LIN {X 0,Y 264.85,Z 561.545,A -85,B 0,C 180,E1 -18192.841,E2 -18192.841} C_VEL
LIN {X 0,Y 265.492,Z 550.133,A -85,B 0,C 180,E1 -18194.761,E2 -18194.761} C_VEL
LIN {X 0,Y 266.161,Z 538.928,A -85,B 0,C 180,E1 -18196.293,E2 -18196.293} C_VEL
LIN {X 0,Y 267.031,Z 524.888,A -85,B 0,C 180,E1 -18197.816,E2 -18197.816} C_VEL
LIN {X 0,Y 267.504,Z 510.963,A -85,B 0,C 180,E1 -18198.948,E2 -18198.948} C_VEL
LIN {X 0,Y 267.86,Z 496.922,A -85,B 0,C 180,E1 -18199.767,E2 -18199.767} C_VEL
LIN {X 0,Y 269.082,Z 449.76,A -85,B 0,C 180,E1 -18201.707,E2 -18201.707} C_VEL
LIN {X 0,Y 269.543,Z 437.735,A -85,B 0,C 180,E1 -18202.197,E2 -18202.197} C_VEL
LIN {X 0,Y 263.446,Z 416.884,A -85,B 0,C 180,E1 -18203.35,E2 -18203.35} C_VEL
LIN {X 0,Y 263.229,Z 415.845,A -85,B 0,C 180,E1 -18203.609,E2 -18203.609} C_VEL
LIN {X 0,Y 263.152,Z 415.684,A -85,B 0,C 180,E1 -18208.197,E2 -18208.197} C_VEL
LIN {X 0,Y 263.129,Z 415.701,A -85,B 0,C 180,E1 -18212.289,E2 -18212.289} C_VEL
LIN {X 0,Y 263.183,Z 415.698,A -85,B 0,C 180,E1 -18216.763,E2 -18216.763} C_VEL
LIN {X 0,Y 263.126,Z 415.699,A -85,B 0,C 180,E1 -18221.594,E2 -18221.594} C_VEL
LIN {X 0,Y 263.161,Z 415.973,A -85,B 0,C 180,E1 -18223.119,E2 -18223.119} C_VEL
LIN {X 0,Y 267.955,Z 428.767,A -85,B 0,C 180,E1 -18227.005,E2 -18227.005} C_VEL
LIN {X 0,Y 272.039,Z 441.377,A -85,B 0,C 180,E1 -18230.442,E2 -18230.442} C_VEL
LIN {X 0,Y 275.291,Z 453.83,A -85,B 0,C 180,E1 -18233.539,E2 -18233.539} C_VEL
LIN {X 0,Y 277.381,Z 463.477,A -85,B 0,C 180,E1 -18235.787,E2 -18235.787} C_VEL
LIN {X 0,Y 277.002,Z 468.199,A -85,B 0,C 180,E1 -18236.672,E2 -18236.672} C_VEL
LIN {X 0,Y 274.845,Z 486.292,A -85,B 0,C 180,E1 -18239.872,E2 -18239.872} C_VEL
LIN {X 0,Y 274.77,Z 488.523,A -85,B 0,C 180,E1 -18240.174,E2 -18240.174} C_VEL
LIN {X 0,Y 279.262,Z 521.145,A -85,B 0,C 180,E1 -18241.646,E2 -18241.646} C_VEL
LIN {X 0,Y 279.718,Z 525.519,A -85,B 0,C 180,E1 -18241.821,E2 -18241.821} C_VEL
LIN {X 0,Y 277.38,Z 599.883,A -85,B 0,C 180,E1 -18243.73,E2 -18243.73} C_VEL
LIN {X 0,Y 276.41,Z 612.805,A -85,B 0,C 180,E1 -18244.289,E2 -18244.289} C_VEL
LIN {X 0,Y 275.09,Z 625.722,A -85,B 0,C 180,E1 -18245.169,E2 -18245.169} C_VEL
LIN {X 0,Y 273.45,Z 638.017,A -85,B 0,C 180,E1 -18246.323,E2 -18246.323} C_VEL
LIN {X 0,Y 271.782,Z 648.339,A -85,B 0,C 180,E1 -18247.578,E2 -18247.578} C_VEL
LIN {X 0,Y 269.838,Z 658.927,A -85,B 0,C 180,E1 -18249.215,E2 -18249.215} C_VEL
LIN {X 0,Y 267.978,Z 668.621,A -85,B 0,C 180,E1 -18251.099,E2 -18251.099} C_VEL
LIN {X 0,Y 266.264,Z 677.005,A -85,B 0,C 180,E1 -18253.122,E2 -18253.122} C_VEL
LIN {X 0,Y 264.551,Z 684.486,A -85,B 0,C 180,E1 -18255.382,E2 -18255.382} C_VEL
LIN {X 0,Y 263.269,Z 690.488,A -85,B 0,C 180,E1 -18257.669,E2 -18257.669} C_VEL
LIN {X 0,Y 262.296,Z 695.236,A -85,B 0,C 180,E1 -18259.97,E2 -18259.97} C_VEL
LIN {X 0,Y 261.682,Z 698.867,A -85,B 0,C 180,E1 -18262.283,E2 -18262.283} C_VEL
LIN {X 0,Y 261.26,Z 701.355,A -85,B 0,C 180,E1 -18264.454,E2 -18264.454} C_VEL
LIN {X 0,Y 261.111,Z 703.163,A -85,B 0,C 180,E1 -18266.914,E2 -18266.914} C_VEL
LIN {X 0,Y 261.076,Z 704.013,A -85,B 0,C 180,E1 -18270,E2 -18270} C_VEL
LIN {X 0,Y 261.054,Z 703.816,A -85,B 0,C 180,E1 -18271.543,E2 -18271.543} C_VEL
LIN {X 0,Y 261.109,Z 703.224,A -85,B 0,C 180,E1 -18273.086,E2 -18273.086} C_VEL
LIN {X 0,Y 261.244,Z 701.499,A -85,B 0,C 180,E1 -18275.509,E2 -18275.509} C_VEL
LIN {X 0,Y 261.808,Z 697.975,A -85,B 0,C 180,E1 -18278.491,E2 -18278.491} C_VEL
LIN {X 0,Y 262.551,Z 694.043,A -85,B 0,C 180,E1 -18280.8,E2 -18280.8} C_VEL
LIN {X 0,Y 263.619,Z 688.947,A -85,B 0,C 180,E1 -18283.098,E2 -18283.098} C_VEL
LIN {X 0,Y 265.02,Z 682.524,A -85,B 0,C 180,E1 -18285.378,E2 -18285.378} C_VEL
LIN {X 0,Y 266.866,Z 674.544,A -85,B 0,C 180,E1 -18287.63,E2 -18287.63} C_VEL
LIN {X 0,Y 268.529,Z 666.026,A -85,B 0,C 180,E1 -18289.575,E2 -18289.575} C_VEL
LIN {X 0,Y 270.323,Z 656.341,A -85,B 0,C 180,E1 -18291.345,E2 -18291.345} C_VEL
LIN {X 0,Y 272.405,Z 645.045,A -85,B 0,C 180,E1 -18292.969,E2 -18292.969} C_VEL
LIN {X 0,Y 274.123,Z 633.931,A -85,B 0,C 180,E1 -18294.218,E2 -18294.218} C_VEL
LIN {X 0,Y 275.628,Z 621.337,A -85,B 0,C 180,E1 -18295.284,E2 -18295.284} C_VEL
LIN {X 0,Y 276.909,Z 608.091,A -85,B 0,C 180,E1 -18296.066,E2 -18296.066} C_VEL
LIN {X 0,Y 277.692,Z 594.677,A -85,B 0,C 180,E1 -18296.542,E2 -18296.542} C_VEL
LIN {X 0,Y 279.693,Z 524.43,A -85,B 0,C 180,E1 -18298.337,E2 -18298.337} C_VEL
LIN {X 0,Y 275.48,Z 492.805,A -85,B 0,C 180,E1 -18299.737,E2 -18299.737} C_VEL
LIN {X 0,Y 274.779,Z 487.724,A -85,B 0,C 180,E1 -18300.016,E2 -18300.016} C_VEL
LIN {X 0,Y 277.378,Z 465.897,A -85,B 0,C 180,E1 -18303.878,E2 -18303.878} C_VEL
LIN {X 0,Y 277.535,Z 464.171,A -85,B 0,C 180,E1 -18304.208,E2 -18304.208} C_VEL
LIN {X 0,Y 275.261,Z 453.468,A -85,B 0,C 180,E1 -18306.688,E2 -18306.688} C_VEL
LIN {X 0,Y 272.521,Z 442.891,A -85,B 0,C 180,E1 -18309.315,E2 -18309.315} C_VEL
LIN {X 0,Y 268.936,Z 431.503,A -85,B 0,C 180,E1 -18312.417,E2 -18312.417} C_VEL
LIN {X 0,Y 265.144,Z 421.282,A -85,B 0,C 180,E1 -18315.379,E2 -18315.379} C_VEL
LIN {X 0,Y 263.143,Z 415.913,A -85,B 0,C 180,E1 -18317.074,E2 -18317.074} C_VEL
LIN {X 0,Y 263.115,Z 415.714,A -85,B 0,C 180,E1 -18320.771,E2 -18320.771} C_VEL
LIN {X 0,Y 263.16,Z 415.701,A -85,B 0,C 180,E1 -18324.017,E2 -18324.017} C_VEL
LIN {X 0,Y 263.111,Z 415.698,A -85,B 0,C 180,E1 -18327.315,E2 -18327.315} C_VEL
LIN {X 0,Y 262.472,Z 415.792,A -85,B 0,C 180,E1 -18328.594,E2 -18328.594} C_VEL
LIN {X 0,Y 259.622,Z 416.159,A -85,B 0,C 180,E1 -18330.677,E2 -18330.677} C_VEL
LIN {X 0,Y 257.197,Z 416.463,A -85,B 0,C 180,E1 -18332.372,E2 -18332.372} C_VEL
LIN {X 0,Y 256.172,Z 416.58,A -85,B 0,C 180,E1 -18333.686,E2 -18333.686} C_VEL
LIN {X 0,Y 256.098,Z 416.584,A -85,B 0,C 180,E1 -18334.132,E2 -18334.132} C_VEL
LIN {X 0,Y 256.074,Z 416.57,A -85,B 0,C 180,E1 -18337.404,E2 -18337.404} C_VEL
LIN {X 0,Y 256.111,Z 416.568,A -85,B 0,C 180,E1 -18340.774,E2 -18340.774} C_VEL
LIN {X 0,Y 256.216,Z 416.56,A -85,B 0,C 180,E1 -18344.08,E2 -18344.08} C_VEL
LIN {X 0,Y 256.277,Z 416.532,A -85,B 0,C 180,E1 -18348.932,E2 -18348.932} C_VEL
LIN {X 0,Y 256.493,Z 416.535,A -85,B 0,C 180,E1 -18352.125,E2 -18352.125} C_VEL
LIN {X 0,Y 256.451,Z 416.518,A -85,B 0,C 180,E1 -18356.858,E2 -18356.858} C_VEL
LIN {X 0,Y 256.699,Z 416.509,A -85,B 0,C 180,E1 -18358.431,E2 -18358.431} C_VEL
LIN {X 0,Y 256.697,Z 416.481,A -85,B 0,C 180,E1 -18361.569,E2 -18361.569} C_VEL
LIN {X 0,Y 256.458,Z 416.539,A -85,B 0,C 180,E1 -18366.293,E2 -18366.293} C_VEL
LIN {X 0,Y 256.405,Z 416.515,A -85,B 0,C 180,E1 -18369.466,E2 -18369.466} C_VEL
LIN {X 0,Y 256.207,Z 416.564,A -85,B 0,C 180,E1 -18374.293,E2 -18374.293} C_VEL
LIN {X 0,Y 256.142,Z 416.553,A -85,B 0,C 180,E1 -18377.567,E2 -18377.567} C_VEL
LIN {X 0,Y 256.121,Z 416.572,A -85,B 0,C 180,E1 -18381.097,E2 -18381.097} C_VEL
LIN {X 0,Y 256.084,Z 416.578,A -85,B 0,C 180,E1 -18385.087,E2 -18385.087} C_VEL
LIN {X 0,Y 256.078,Z 416.564,A -85,B 0,C 180,E1 -18388.569,E2 -18388.569} C_VEL
LIN {X 0,Y 256.072,Z 416.588,A -85,B 0,C 180,E1 -18391.699,E2 -18391.699} C_VEL
LIN {X 0,Y 256.081,Z 416.57,A -85,B 0,C 180,E1 -18395.193,E2 -18395.193} C_VEL
LIN {X 0,Y 256.107,Z 416.584,A -85,B 0,C 180,E1 -18397.268,E2 -18397.268} C_VEL
LIN {X 0,Y 256.018,Z 416.527,A -85,B 0,C 180,E1 -18401.211,E2 -18401.211} C_VEL
LIN {X 0,Y 256.034,Z 416.594,A -85,B 0,C 180,E1 -18405.536,E2 -18405.536} C_VEL
LIN {X 0,Y 256.023,Z 416.717,A -85,B 0,C 180,E1 -18409.354,E2 -18409.354} C_VEL
LIN {X 0,Y 256.297,Z 417.843,A -85,B 0,C 180,E1 -18409.759,E2 -18409.759} C_VEL
LIN {X 0,Y 259.881,Z 424.387,A -85,B 0,C 180,E1 -18411.31,E2 -18411.31} C_VEL
LIN {X 0,Y 263.321,Z 435.836,A -85,B 0,C 180,E1 -18413.197,E2 -18413.197} C_VEL
LIN {X 0,Y 267.896,Z 451.956,A -85,B 0,C 180,E1 -18415.612,E2 -18415.612} C_VEL
LIN {X 0,Y 268.711,Z 455.376,A -85,B 0,C 180,E1 -18416.083,E2 -18416.083} C_VEL
LIN {X 0,Y 268.725,Z 480.622,A -85,B 0,C 180,E1 -18418.681,E2 -18418.681} C_VEL
LIN {X 0,Y 268.671,Z 489.032,A -85,B 0,C 180,E1 -18419.496,E2 -18419.496} C_VEL
LIN {X 0,Y 271.982,Z 520.346,A -85,B 0,C 180,E1 -18420.837,E2 -18420.837} C_VEL
LIN {X 0,Y 272.827,Z 533.578,A -85,B 0,C 180,E1 -18421.325,E2 -18421.325} C_VEL
LIN {X 0,Y 270.595,Z 602.971,A -85,B 0,C 180,E1 -18423.122,E2 -18423.122} C_VEL
LIN {X 0,Y 269.625,Z 616.536,A -85,B 0,C 180,E1 -18423.697,E2 -18423.697} C_VEL
LIN {X 0,Y 268.323,Z 628.565,A -85,B 0,C 180,E1 -18424.498,E2 -18424.498} C_VEL
LIN {X 0,Y 266.64,Z 641.245,A -85,B 0,C 180,E1 -18425.679,E2 -18425.679} C_VEL
LIN {X 0,Y 264.897,Z 651.794,A -85,B 0,C 180,E1 -18426.962,E2 -18426.962} C_VEL
LIN {X 0,Y 262.808,Z 662.552,A -85,B 0,C 180,E1 -18428.631,E2 -18428.631} C_VEL
LIN {X 0,Y 260.829,Z 672.425,A -85,B 0,C 180,E1 -18430.574,E2 -18430.574} C_VEL
LIN {X 0,Y 259.036,Z 680.818,A -85,B 0,C 180,E1 -18432.635,E2 -18432.635} C_VEL
LIN {X 0,Y 257.333,Z 688.353,A -85,B 0,C 180,E1 -18434.962,E2 -18434.962} C_VEL
LIN {X 0,Y 256.017,Z 694.402,A -85,B 0,C 180,E1 -18437.314,E2 -18437.314} C_VEL
LIN {X 0,Y 255.09,Z 699.178,A -85,B 0,C 180,E1 -18439.683,E2 -18439.683} C_VEL
LIN {X 0,Y 254.443,Z 702.823,A -85,B 0,C 180,E1 -18442.061,E2 -18442.061} C_VEL
LIN {X 0,Y 254.126,Z 705.608,A -85,B 0,C 180,E1 -18444.625,E2 -18444.625} C_VEL
LIN {X 0,Y 254.03,Z 707.114,A -85,B 0,C 180,E1 -18446.828,E2 -18446.828} C_VEL
LIN {X 0,Y 254.025,Z 707.724,A -85,B 0,C 180,E1 -18448.414,E2 -18448.414} C_VEL
LIN {X 0,Y 254.065,Z 707.939,A -85,B 0,C 180,E1 -18450,E2 -18450} C_VEL
LIN {X 0,Y 254.067,Z 707.715,A -85,B 0,C 180,E1 -18451.585,E2 -18451.585} C_VEL
LIN {X 0,Y 254.054,Z 707.099,A -85,B 0,C 180,E1 -18453.171,E2 -18453.171} C_VEL
LIN {X 0,Y 254.134,Z 705.563,A -85,B 0,C 180,E1 -18455.394,E2 -18455.394} C_VEL
LIN {X 0,Y 254.451,Z 702.782,A -85,B 0,C 180,E1 -18457.938,E2 -18457.938} C_VEL
LIN {X 0,Y 255.092,Z 699.121,A -85,B 0,C 180,E1 -18460.316,E2 -18460.316} C_VEL
LIN {X 0,Y 256.021,Z 694.331,A -85,B 0,C 180,E1 -18462.686,E2 -18462.686} C_VEL
LIN {X 0,Y 257.345,Z 688.269,A -85,B 0,C 180,E1 -18465.037,E2 -18465.037} C_VEL
LIN {X 0,Y 259.024,Z 680.707,A -85,B 0,C 180,E1 -18467.365,E2 -18467.365} C_VEL
LIN {X 0,Y 260.837,Z 672.247,A -85,B 0,C 180,E1 -18469.431,E2 -18469.431} C_VEL
LIN {X 0,Y 262.817,Z 662.368,A -85,B 0,C 180,E1 -18471.367,E2 -18471.367} C_VEL
LIN {X 0,Y 264.865,Z 651.56,A -85,B 0,C 180,E1 -18473.04,E2 -18473.04} C_VEL
LIN {X 0,Y 266.889,Z 639.21,A -85,B 0,C 180,E1 -18474.503,E2 -18474.503} C_VEL
LIN {X 0,Y 267.731,Z 633.457,A -85,B 0,C 180,E1 -18475.094,E2 -18475.094} C_VEL
LIN {X 0,Y 272.517,Z 622.346,A -85,B 0,C 180,E1 -18477.243,E2 -18477.243} C_VEL
LIN {X 0,Y 277.231,Z 610.736,A -85,B 0,C 180,E1 -18479.001,E2 -18479.001} C_VEL
LIN {X 0,Y 281.94,Z 597.942,A -85,B 0,C 180,E1 -18480.524,E2 -18480.524} C_VEL
LIN {X 0,Y 285.924,Z 585.491,A -85,B 0,C 180,E1 -18481.695,E2 -18481.695} C_VEL
LIN {X 0,Y 289.914,Z 571.079,A -85,B 0,C 180,E1 -18482.744,E2 -18482.744} C_VEL
LIN {X 0,Y 293.532,Z 553.924,A -85,B 0,C 180,E1 -18483.688,E2 -18483.688} C_VEL
LIN {X 0,Y 296.227,Z 535.792,A -85,B 0,C 180,E1 -18484.52,E2 -18484.52} C_VEL
LIN {X 0,Y 297.419,Z 522.403,A -85,B 0,C 180,E1 -18485.437,E2 -18485.437} C_VEL
LIN {X 0,Y 298.17,Z 508.364,A -85,B 0,C 180,E1 -18486.705,E2 -18486.705} C_VEL
LIN {X 0,Y 298.597,Z 495.67,A -85,B 0,C 180,E1 -18488.12,E2 -18488.12} C_VEL
LIN {X 0,Y 298.719,Z 489.21,A -85,B 0,C 180,E1 -18488.995,E2 -18488.995} C_VEL
LIN {X 0,Y 297.581,Z 483.469,A -85,B 0,C 180,E1 -18490.746,E2 -18490.746} C_VEL
LIN {X 0,Y 296.387,Z 477.666,A -85,B 0,C 180,E1 -18493.445,E2 -18493.445} C_VEL
LIN {X 0,Y 296.175,Z 474.72,A -85,B 0,C 180,E1 -18495.573,E2 -18495.573} C_VEL
LIN {X 0,Y 296.767,Z 472.828,A -85,B 0,C 180,E1 -18498.053,E2 -18498.053} C_VEL
LIN {X 0,Y 298.296,Z 472.538,A -85,B 0,C 180,E1 -18500.496,E2 -18500.496} C_VEL
LIN {X 0,Y 300.271,Z 473.517,A -85,B 0,C 180,E1 -18502.516,E2 -18502.516} C_VEL
LIN {X 0,Y 302.602,Z 475.847,A -85,B 0,C 180,E1 -18504.379,E2 -18504.379} C_VEL
LIN {X 0,Y 304.246,Z 477.887,A -85,B 0,C 180,E1 -18505.466,E2 -18505.466} C_VEL
LIN {X 0,Y 299.441,Z 507.153,A -85,B 0,C 180,E1 -18506.881,E2 -18506.881} C_VEL
LIN {X 0,Y 297.506,Z 521.717,A -85,B 0,C 180,E1 -18507.742,E2 -18507.742} C_VEL
LIN {X 0,Y 295.036,Z 535.372,A -85,B 0,C 180,E1 -18508.795,E2 -18508.795} C_VEL
LIN {X 0,Y 292.316,Z 546.909,A -85,B 0,C 180,E1 -18509.944,E2 -18509.944} C_VEL
LIN {X 0,Y 289.223,Z 557.964,A -85,B 0,C 180,E1 -18511.32,E2 -18511.32} C_VEL
LIN {X 0,Y 285.591,Z 568.323,A -85,B 0,C 180,E1 -18512.918,E2 -18512.918} C_VEL
LIN {X 0,Y 282.305,Z 576.824,A -85,B 0,C 180,E1 -18514.535,E2 -18514.535} C_VEL
LIN {X 0,Y 278.49,Z 585.306,A -85,B 0,C 180,E1 -18516.58,E2 -18516.58} C_VEL
LIN {X 0,Y 274.934,Z 592.143,A -85,B 0,C 180,E1 -18518.638,E2 -18518.638} C_VEL
LIN {X 0,Y 271.125,Z 598.395,A -85,B 0,C 180,E1 -18521.094,E2 -18521.094} C_VEL
LIN {X 0,Y 267.32,Z 603.574,A -85,B 0,C 180,E1 -18523.975,E2 -18523.975} C_VEL
LIN {X 0,Y 264.813,Z 606.237,A -85,B 0,C 180,E1 -18526.181,E2 -18526.181} C_VEL
LIN {X 0,Y 263.333,Z 607.422,A -85,B 0,C 180,E1 -18527.672,E2 -18527.672} C_VEL
LIN {X 0,Y 260.7,Z 608.594,A -85,B 0,C 180,E1 -18530.692,E2 -18530.692} C_VEL
LIN {X 0,Y 259.67,Z 608.534,A -85,B 0,C 180,E1 -18532.223,E2 -18532.223} C_VEL
LIN {X 0,Y 258.912,Z 608.014,A -85,B 0,C 180,E1 -18533.767,E2 -18533.767} C_VEL
LIN {X 0,Y 258.281,Z 607.095,A -85,B 0,C 180,E1 -18535.318,E2 -18535.318} C_VEL
LIN {X 0,Y 257.555,Z 605.796,A -85,B 0,C 180,E1 -18536.872,E2 -18536.872} C_VEL
LIN {X 0,Y 256.743,Z 602.999,A -85,B 0,C 180,E1 -18539.216,E2 -18539.216} C_VEL
LIN {X 0,Y 256.327,Z 599.154,A -85,B 0,C 180,E1 -18541.571,E2 -18541.571} C_VEL
LIN {X 0,Y 256.161,Z 594.186,A -85,B 0,C 180,E1 -18543.933,E2 -18543.933} C_VEL
LIN {X 0,Y 256.322,Z 586.806,A -85,B 0,C 180,E1 -18546.692,E2 -18546.692} C_VEL
LIN {X 0,Y 256.735,Z 578.927,A -85,B 0,C 180,E1 -18549.056,E2 -18549.056} C_VEL
LIN {X 0,Y 257.298,Z 569.105,A -85,B 0,C 180,E1 -18551.422,E2 -18551.422} C_VEL
LIN {X 0,Y 257.907,Z 559.145,A -85,B 0,C 180,E1 -18553.393,E2 -18553.393} C_VEL
LIN {X 0,Y 258.623,Z 546.833,A -85,B 0,C 180,E1 -18555.364,E2 -18555.364} C_VEL
LIN {X 0,Y 259.376,Z 534.597,A -85,B 0,C 180,E1 -18556.935,E2 -18556.935} C_VEL
LIN {X 0,Y 260.126,Z 521.014,A -85,B 0,C 180,E1 -18558.305,E2 -18558.305} C_VEL
LIN {X 0,Y 260.522,Z 507.02,A -85,B 0,C 180,E1 -18559.361,E2 -18559.361} C_VEL
LIN {X 0,Y 260.898,Z 492.906,A -85,B 0,C 180,E1 -18560.109,E2 -18560.109} C_VEL
LIN {X 0,Y 262.036,Z 451.118,A -85,B 0,C 180,E1 -18561.899,E2 -18561.899} C_VEL
LIN {X 0,Y 262.46,Z 438.689,A -85,B 0,C 180,E1 -18562.423,E2 -18562.423} C_VEL
LIN {X 0,Y 256.376,Z 417.606,A -85,B 0,C 180,E1 -18563.616,E2 -18563.616} C_VEL
LIN {X 0,Y 256.189,Z 416.651,A -85,B 0,C 180,E1 -18563.928,E2 -18563.928} C_VEL
LIN {X 0,Y 256.094,Z 416.561,A -85,B 0,C 180,E1 -18568.577,E2 -18568.577} C_VEL
LIN {X 0,Y 256.076,Z 416.588,A -85,B 0,C 180,E1 -18571.702,E2 -18571.702} C_VEL
LIN {X 0,Y 256.083,Z 416.575,A -85,B 0,C 180,E1 -18575.193,E2 -18575.193} C_VEL
LIN {X 0,Y 256.115,Z 416.572,A -85,B 0,C 180,E1 -18577.271,E2 -18577.271} C_VEL
LIN {X 0,Y 256.129,Z 416.804,A -85,B 0,C 180,E1 -18581.83,E2 -18581.83} C_VEL
LIN {X 0,Y 260.412,Z 428.088,A -85,B 0,C 180,E1 -18585.437,E2 -18585.437} C_VEL
LIN {X 0,Y 263.748,Z 437.752,A -85,B 0,C 180,E1 -18588.255,E2 -18588.255} C_VEL
LIN {X 0,Y 266.799,Z 447.885,A -85,B 0,C 180,E1 -18590.994,E2 -18590.994} C_VEL
LIN {X 0,Y 269.972,Z 460.995,A -85,B 0,C 180,E1 -18594.251,E2 -18594.251} C_VEL
LIN {X 0,Y 270.983,Z 466.791,A -85,B 0,C 180,E1 -18595.577,E2 -18595.577} C_VEL
LIN {X 0,Y 268.545,Z 486.331,A -85,B 0,C 180,E1 -18599.096,E2 -18599.096} C_VEL
LIN {X 0,Y 268.429,Z 488.341,A -85,B 0,C 180,E1 -18599.388,E2 -18599.388} C_VEL
LIN {X 0,Y 273.023,Z 521.924,A -85,B 0,C 180,E1 -18600.961,E2 -18600.961} C_VEL
LIN {X 0,Y 273.425,Z 527.263,A -85,B 0,C 180,E1 -18601.165,E2 -18601.165} C_VEL
LIN {X 0,Y 270.974,Z 601.199,A -85,B 0,C 180,E1 -18603.111,E2 -18603.111} C_VEL
LIN {X 0,Y 269.893,Z 614.342,A -85,B 0,C 180,E1 -18603.725,E2 -18603.725} C_VEL
LIN {X 0,Y 268.431,Z 627.911,A -85,B 0,C 180,E1 -18604.717,E2 -18604.717} C_VEL
LIN {X 0,Y 266.728,Z 639.694,A -85,B 0,C 180,E1 -18605.895,E2 -18605.895} C_VEL
LIN {X 0,Y 264.759,Z 650.917,A -85,B 0,C 180,E1 -18607.362,E2 -18607.362} C_VEL
LIN {X 0,Y 262.814,Z 661.059,A -85,B 0,C 180,E1 -18609.043,E2 -18609.043} C_VEL
LIN {X 0,Y 260.802,Z 671.014,A -85,B 0,C 180,E1 -18611.133,E2 -18611.133} C_VEL
LIN {X 0,Y 258.816,Z 679.726,A -85,B 0,C 180,E1 -18613.434,E2 -18613.434} C_VEL
LIN {X 0,Y 257.152,Z 686.717,A -85,B 0,C 180,E1 -18615.761,E2 -18615.761} C_VEL
LIN {X 0,Y 255.936,Z 692.271,A -85,B 0,C 180,E1 -18618.115,E2 -18618.115} C_VEL
LIN {X 0,Y 255.028,Z 696.629,A -85,B 0,C 180,E1 -18620.483,E2 -18620.483} C_VEL
LIN {X 0,Y 254.627,Z 698.922,A -85,B 0,C 180,E1 -18622.068,E2 -18622.068} C_VEL
LIN {X 0,Y 254.168,Z 701.613,A -85,B 0,C 180,E1 -18624.526,E2 -18624.526} C_VEL
LIN {X 0,Y 254.012,Z 703.218,A -85,B 0,C 180,E1 -18626.828,E2 -18626.828} C_VEL
LIN {X 0,Y 253.967,Z 703.833,A -85,B 0,C 180,E1 -18628.414,E2 -18628.414} C_VEL
LIN {X 0,Y 253.984,Z 704.067,A -85,B 0,C 180,E1 -18630,E2 -18630} C_VEL
LIN {X 0,Y 253.966,Z 703.87,A -85,B 0,C 180,E1 -18631.586,E2 -18631.586} C_VEL
LIN {X 0,Y 254.01,Z 703.278,A -85,B 0,C 180,E1 -18633.172,E2 -18633.172} C_VEL
LIN {X 0,Y 254.135,Z 701.794,A -85,B 0,C 180,E1 -18635.394,E2 -18635.394} C_VEL
LIN {X 0,Y 254.564,Z 699.081,A -85,B 0,C 180,E1 -18637.935,E2 -18637.935} C_VEL
LIN {X 0,Y 255.267,Z 695.504,A -85,B 0,C 180,E1 -18640.309,E2 -18640.309} C_VEL
LIN {X 0,Y 256.273,Z 690.812,A -85,B 0,C 180,E1 -18642.674,E2 -18642.674} C_VEL
LIN {X 0,Y 257.587,Z 684.867,A -85,B 0,C 180,E1 -18645.023,E2 -18645.023} C_VEL
LIN {X 0,Y 259.401,Z 677.47,A -85,B 0,C 180,E1 -18647.339,E2 -18647.339} C_VEL
LIN {X 0,Y 261.344,Z 668.537,A -85,B 0,C 180,E1 -18649.557,E2 -18649.557} C_VEL
LIN {X 0,Y 263.281,Z 658.574,A -85,B 0,C 180,E1 -18651.534,E2 -18651.534} C_VEL
LIN {X 0,Y 265.401,Z 647.843,A -85,B 0,C 180,E1 -18653.198,E2 -18653.198} C_VEL
LIN {X 0,Y 267.435,Z 635.686,A -85,B 0,C 180,E1 -18654.657,E2 -18654.657} C_VEL
LIN {X 0,Y 268.983,Z 623.804,A -85,B 0,C 180,E1 -18655.746,E2 -18655.746} C_VEL
LIN {X 0,Y 270.248,Z 611.484,A -85,B 0,C 180,E1 -18656.55,E2 -18656.55} C_VEL
LIN {X 0,Y 271.224,Z 597.771,A -85,B 0,C 180,E1 -18657.123,E2 -18657.123} C_VEL
LIN {X 0,Y 273.395,Z 524.791,A -85,B 0,C 180,E1 -18659.038,E2 -18659.038} C_VEL
LIN {X 0,Y 269.172,Z 492.941,A -85,B 0,C 180,E1 -18660.5,E2 -18660.5} C_VEL
LIN {X 0,Y 268.473,Z 487.826,A -85,B 0,C 180,E1 -18660.779,E2 -18660.779} C_VEL
LIN {X 0,Y 270.976,Z 467.525,A -85,B 0,C 180,E1 -18664.418,E2 -18664.418} C_VEL
LIN {X 0,Y 270.801,Z 464.663,A -85,B 0,C 180,E1 -18665.044,E2 -18665.044} C_VEL
LIN {X 0,Y 267.934,Z 452.006,A -85,B 0,C 180,E1 -18668.102,E2 -18668.102} C_VEL
LIN {X 0,Y 265.472,Z 443.079,A -85,B 0,C 180,E1 -18670.437,E2 -18670.437} C_VEL
LIN {X 0,Y 261.856,Z 431.948,A -85,B 0,C 180,E1 -18673.559,E2 -18673.559} C_VEL
LIN {X 0,Y 257.599,Z 420.812,A -85,B 0,C 180,E1 -18676.994,E2 -18676.994} C_VEL
LIN {X 0,Y 256.112,Z 416.811,A -85,B 0,C 180,E1 -18678.33,E2 -18678.33} C_VEL
LIN {X 0,Y 256.068,Z 416.592,A -85,B 0,C 180,E1 -18680.857,E2 -18680.857} C_VEL
LIN {X 0,Y 256.082,Z 416.587,A -85,B 0,C 180,E1 -18684.807,E2 -18684.807} C_VEL
LIN {X 0,Y 256.08,Z 416.589,A -85,B 0,C 180,E1 -18688.57,E2 -18688.57} C_VEL
LIN {X 0,Y 256.088,Z 416.573,A -85,B 0,C 180,E1 -18692.19,E2 -18692.19} C_VEL
LIN {X 0,Y 256.098,Z 416.584,A -85,B 0,C 180,E1 -18694.132,E2 -18694.132} C_VEL
LIN {X 0,Y 255.446,Z 416.652,A -85,B 0,C 180,E1 -18695.445,E2 -18695.445} C_VEL
LIN {X 0,Y 252.574,Z 417.011,A -85,B 0,C 180,E1 -18697.585,E2 -18697.585} C_VEL
LIN {X 0,Y 250.136,Z 417.329,A -85,B 0,C 180,E1 -18699.328,E2 -18699.328} C_VEL
LIN {X 0,Y 249.111,Z 417.441,A -85,B 0,C 180,E1 -18700.68,E2 -18700.68} C_VEL
LIN {X 0,Y 249.039,Z 417.444,A -85,B 0,C 180,E1 -18701.138,E2 -18701.138} C_VEL
LIN {X 0,Y 249.16,Z 417.432,A -85,B 0,C 180,E1 -18703.616,E2 -18703.616} C_VEL
LIN {X 0,Y 249.222,Z 417.41,A -85,B 0,C 180,E1 -18708.615,E2 -18708.615} C_VEL
LIN {X 0,Y 249.434,Z 417.416,A -85,B 0,C 180,E1 -18711.901,E2 -18711.901} C_VEL
LIN {X 0,Y 249.261,Z 417.404,A -85,B 0,C 180,E1 -18715.148,E2 -18715.148} C_VEL
LIN {X 0,Y 249.66,Z 417.385,A -85,B 0,C 180,E1 -18718.387,E2 -18718.387} C_VEL
LIN {X 0,Y 249.658,Z 417.357,A -85,B 0,C 180,E1 -18721.613,E2 -18721.613} C_VEL
LIN {X 0,Y 249.429,Z 417.414,A -85,B 0,C 180,E1 -18726.471,E2 -18726.471} C_VEL
LIN {X 0,Y 249.335,Z 417.395,A -85,B 0,C 180,E1 -18729.737,E2 -18729.737} C_VEL
LIN {X 0,Y 249.151,Z 417.435,A -85,B 0,C 180,E1 -18734.707,E2 -18734.707} C_VEL
LIN {X 0,Y 249.075,Z 417.439,A -85,B 0,C 180,E1 -18738.082,E2 -18738.082} C_VEL
LIN {X 0,Y 249.045,Z 417.447,A -85,B 0,C 180,E1 -18741.522,E2 -18741.522} C_VEL
LIN {X 0,Y 249.046,Z 417.46,A -85,B 0,C 180,E1 -18745.439,E2 -18745.439} C_VEL
LIN {X 0,Y 249.026,Z 417.441,A -85,B 0,C 180,E1 -18748.968,E2 -18748.968} C_VEL
LIN {X 0,Y 249.028,Z 417.463,A -85,B 0,C 180,E1 -18752.426,E2 -18752.426} C_VEL
LIN {X 0,Y 249.026,Z 417.462,A -85,B 0,C 180,E1 -18756.346,E2 -18756.346} C_VEL
LIN {X 0,Y 248.98,Z 417.406,A -85,B 0,C 180,E1 -18760.483,E2 -18760.483} C_VEL
LIN {X 0,Y 248.974,Z 417.46,A -85,B 0,C 180,E1 -18764.886,E2 -18764.886} C_VEL
LIN {X 0,Y 248.999,Z 417.602,A -85,B 0,C 180,E1 -18767.873,E2 -18767.873} C_VEL
LIN {X 0,Y 249.306,Z 418.897,A -85,B 0,C 180,E1 -18768.334,E2 -18768.334} C_VEL
LIN {X 0,Y 251.061,Z 421.666,A -85,B 0,C 180,E1 -18769.097,E2 -18769.097} C_VEL
LIN {X 0,Y 255.051,Z 429.466,A -85,B 0,C 180,E1 -18770.929,E2 -18770.929} C_VEL
LIN {X 0,Y 259.7,Z 445.846,A -85,B 0,C 180,E1 -18773.62,E2 -18773.62} C_VEL
LIN {X 0,Y 262.755,Z 458.031,A -85,B 0,C 180,E1 -18775.446,E2 -18775.446} C_VEL
LIN {X 0,Y 262.591,Z 480.771,A -85,B 0,C 180,E1 -18777.863,E2 -18777.863} C_VEL
LIN {X 0,Y 262.412,Z 488.754,A -85,B 0,C 180,E1 -18778.675,E2 -18778.675} C_VEL
LIN {X 0,Y 265.633,Z 519.132,A -85,B 0,C 180,E1 -18780.03,E2 -18780.03} C_VEL
LIN {X 0,Y 266.643,Z 533.45,A -85,B 0,C 180,E1 -18780.589,E2 -18780.589} C_VEL
LIN {X 0,Y 264.358,Z 601.599,A -85,B 0,C 180,E1 -18782.381,E2 -18782.381} C_VEL
LIN {X 0,Y 263.48,Z 614.792,A -85,B 0,C 180,E1 -18782.927,E2 -18782.927} C_VEL
LIN {X 0,Y 262.075,Z 627.433,A -85,B 0,C 180,E1 -18783.738,E2 -18783.738} C_VEL
LIN {X 0,Y 260.441,Z 639.476,A -85,B 0,C 180,E1 -18784.848,E2 -18784.848} C_VEL
LIN {X 0,Y 258.377,Z 651.757,A -85,B 0,C 180,E1 -18786.346,E2 -18786.346} C_VEL
LIN {X 0,Y 256.198,Z 662.51,A -85,B 0,C 180,E1 -18788.052,E2 -18788.052} C_VEL
LIN {X 0,Y 254.27,Z 671.625,A -85,B 0,C 180,E1 -18789.872,E2 -18789.872} C_VEL
LIN {X 0,Y 252.23,Z 680.769,A -85,B 0,C 180,E1 -18792.151,E2 -18792.151} C_VEL
LIN {X 0,Y 250.482,Z 688.303,A -85,B 0,C 180,E1 -18794.541,E2 -18794.541} C_VEL
LIN {X 0,Y 249.05,Z 694.351,A -85,B 0,C 180,E1 -18796.952,E2 -18796.952} C_VEL
LIN {X 0,Y 248.088,Z 699.126,A -85,B 0,C 180,E1 -18799.389,E2 -18799.389} C_VEL
LIN {X 0,Y 247.395,Z 702.77,A -85,B 0,C 180,E1 -18801.834,E2 -18801.834} C_VEL
LIN {X 0,Y 247.023,Z 705.789,A -85,B 0,C 180,E1 -18804.736,E2 -18804.736} C_VEL
LIN {X 0,Y 246.931,Z 707.06,A -85,B 0,C 180,E1 -18806.737,E2 -18806.737} C_VEL
LIN {X 0,Y 246.935,Z 707.67,A -85,B 0,C 180,E1 -18808.369,E2 -18808.369} C_VEL
LIN {X 0,Y 246.971,Z 707.885,A -85,B 0,C 180,E1 -18810,E2 -18810} C_VEL
LIN {X 0,Y 246.974,Z 707.661,A -85,B 0,C 180,E1 -18811.63,E2 -18811.63} C_VEL
LIN {X 0,Y 246.955,Z 707.045,A -85,B 0,C 180,E1 -18813.263,E2 -18813.263} C_VEL
LIN {X 0,Y 247.022,Z 705.761,A -85,B 0,C 180,E1 -18815.264,E2 -18815.264} C_VEL
LIN {X 0,Y 247.402,Z 702.727,A -85,B 0,C 180,E1 -18818.166,E2 -18818.166} C_VEL
LIN {X 0,Y 248.089,Z 699.067,A -85,B 0,C 180,E1 -18820.611,E2 -18820.611} C_VEL
LIN {X 0,Y 249.055,Z 694.277,A -85,B 0,C 180,E1 -18823.047,E2 -18823.047} C_VEL
LIN {X 0,Y 250.493,Z 688.216,A -85,B 0,C 180,E1 -18825.458,E2 -18825.458} C_VEL
LIN {X 0,Y 252.22,Z 680.655,A -85,B 0,C 180,E1 -18827.849,E2 -18827.849} C_VEL
LIN {X 0,Y 253.989,Z 672.879,A -85,B 0,C 180,E1 -18829.814,E2 -18829.814} C_VEL
LIN {X 0,Y 255.966,Z 663.377,A -85,B 0,C 180,E1 -18831.757,E2 -18831.757} C_VEL
LIN {X 0,Y 258.07,Z 652.833,A -85,B 0,C 180,E1 -18833.471,E2 -18833.471} C_VEL
LIN {X 0,Y 259.902,Z 642.618,A -85,B 0,C 180,E1 -18834.78,E2 -18834.78} C_VEL
LIN {X 0,Y 261.112,Z 635.111,A -85,B 0,C 180,E1 -18835.616,E2 -18835.616} C_VEL
LIN {X 0,Y 265.489,Z 625.87,A -85,B 0,C 180,E1 -18837.598,E2 -18837.598} C_VEL
LIN {X 0,Y 270.721,Z 614.318,A -85,B 0,C 180,E1 -18839.554,E2 -18839.554} C_VEL
LIN {X 0,Y 276.012,Z 601.403,A -85,B 0,C 180,E1 -18841.252,E2 -18841.252} C_VEL
LIN {X 0,Y 280.61,Z 588.566,A -85,B 0,C 180,E1 -18842.58,E2 -18842.58} C_VEL
LIN {X 0,Y 285.051,Z 574.481,A -85,B 0,C 180,E1 -18843.693,E2 -18843.693} C_VEL
LIN {X 0,Y 288.633,Z 560.138,A -85,B 0,C 180,E1 -18844.586,E2 -18844.586} C_VEL
LIN {X 0,Y 291.802,Z 543.136,A -85,B 0,C 180,E1 -18845.401,E2 -18845.401} C_VEL
LIN {X 0,Y 293.012,Z 534.6,A -85,B 0,C 180,E1 -18845.853,E2 -18845.853} C_VEL
LIN {X 0,Y 294.112,Z 523.656,A -85,B 0,C 180,E1 -18846.652,E2 -18846.652} C_VEL
LIN {X 0,Y 295.115,Z 510.228,A -85,B 0,C 180,E1 -18847.902,E2 -18847.902} C_VEL
LIN {X 0,Y 295.84,Z 497.661,A -85,B 0,C 180,E1 -18849.365,E2 -18849.365} C_VEL
LIN {X 0,Y 295.986,Z 494.154,A -85,B 0,C 180,E1 -18849.874,E2 -18849.874} C_VEL
LIN {X 0,Y 295.242,Z 489.342,A -85,B 0,C 180,E1 -18851.382,E2 -18851.382} C_VEL
LIN {X 0,Y 294.433,Z 484.047,A -85,B 0,C 180,E1 -18853.915,E2 -18853.915} C_VEL
LIN {X 0,Y 294.408,Z 481.149,A -85,B 0,C 180,E1 -18856.118,E2 -18856.118} C_VEL
LIN {X 0,Y 295.142,Z 479.595,A -85,B 0,C 180,E1 -18858.405,E2 -18858.405} C_VEL
LIN {X 0,Y 296.688,Z 479.482,A -85,B 0,C 180,E1 -18860.733,E2 -18860.733} C_VEL
LIN {X 0,Y 298.372,Z 480.383,A -85,B 0,C 180,E1 -18862.449,E2 -18862.449} C_VEL
LIN {X 0,Y 300.407,Z 482.463,A -85,B 0,C 180,E1 -18864.139,E2 -18864.139} C_VEL
LIN {X 0,Y 300.765,Z 483.042,A -85,B 0,C 180,E1 -18864.427,E2 -18864.427} C_VEL
LIN {X 0,Y 295.857,Z 511.865,A -85,B 0,C 180,E1 -18865.861,E2 -18865.861} C_VEL
LIN {X 0,Y 293.588,Z 526.476,A -85,B 0,C 180,E1 -18866.798,E2 -18866.798} C_VEL
LIN {X 0,Y 290.397,Z 541.359,A -85,B 0,C 180,E1 -18868.035,E2 -18868.035} C_VEL
LIN {X 0,Y 287.206,Z 553.112,A -85,B 0,C 180,E1 -18869.352,E2 -18869.352} C_VEL
LIN {X 0,Y 283.277,Z 564.76,A -85,B 0,C 180,E1 -18870.965,E2 -18870.965} C_VEL
LIN {X 0,Y 279.306,Z 574.766,A -85,B 0,C 180,E1 -18872.706,E2 -18872.706} C_VEL
LIN {X 0,Y 275.205,Z 583.611,A -85,B 0,C 180,E1 -18874.675,E2 -18874.675} C_VEL
LIN {X 0,Y 271.325,Z 591.001,A -85,B 0,C 180,E1 -18876.733,E2 -18876.733} C_VEL
LIN {X 0,Y 268.258,Z 596.009,A -85,B 0,C 180,E1 -18878.483,E2 -18878.483} C_VEL
LIN {X 0,Y 264.829,Z 600.935,A -85,B 0,C 180,E1 -18880.627,E2 -18880.627} C_VEL
LIN {X 0,Y 261.76,Z 604.697,A -85,B 0,C 180,E1 -18882.822,E2 -18882.822} C_VEL
LIN {X 0,Y 259.849,Z 606.622,A -85,B 0,C 180,E1 -18884.308,E2 -18884.308} C_VEL
LIN {X 0,Y 256.601,Z 609.122,A -85,B 0,C 180,E1 -18887.343,E2 -18887.343} C_VEL
LIN {X 0,Y 255.145,Z 609.768,A -85,B 0,C 180,E1 -18888.883,E2 -18888.883} C_VEL
LIN {X 0,Y 253.851,Z 609.953,A -85,B 0,C 180,E1 -18890.438,E2 -18890.438} C_VEL
LIN {X 0,Y 252.745,Z 609.724,A -85,B 0,C 180,E1 -18892.008,E2 -18892.008} C_VEL
LIN {X 0,Y 251.951,Z 609.074,A -85,B 0,C 180,E1 -18893.594,E2 -18893.594} C_VEL
LIN {X 0,Y 251.276,Z 608.004,A -85,B 0,C 180,E1 -18895.187,E2 -18895.187} C_VEL
LIN {X 0,Y 250.522,Z 606.518,A -85,B 0,C 180,E1 -18896.784,E2 -18896.784} C_VEL
LIN {X 0,Y 249.681,Z 603.482,A -85,B 0,C 180,E1 -18899.194,E2 -18899.194} C_VEL
LIN {X 0,Y 249.231,Z 599.411,A -85,B 0,C 180,E1 -18901.616,E2 -18901.616} C_VEL
LIN {X 0,Y 249.048,Z 593.207,A -85,B 0,C 180,E1 -18904.451,E2 -18904.451} C_VEL
LIN {X 0,Y 249.253,Z 586.455,A -85,B 0,C 180,E1 -18906.883,E2 -18906.883} C_VEL
LIN {X 0,Y 249.678,Z 578.169,A -85,B 0,C 180,E1 -18909.315,E2 -18909.315} C_VEL
LIN {X 0,Y 250.174,Z 569.841,A -85,B 0,C 180,E1 -18911.341,E2 -18911.341} C_VEL
LIN {X 0,Y 250.841,Z 558.704,A -85,B 0,C 180,E1 -18913.571,E2 -18913.571} C_VEL
LIN {X 0,Y 251.493,Z 547.48,A -85,B 0,C 180,E1 -18915.396,E2 -18915.396} C_VEL
LIN {X 0,Y 252.276,Z 535.112,A -85,B 0,C 180,E1 -18917.009,E2 -18917.009} C_VEL
LIN {X 0,Y 253.059,Z 521.396,A -85,B 0,C 180,E1 -18918.416,E2 -18918.416} C_VEL
LIN {X 0,Y 253.527,Z 505.948,A -85,B 0,C 180,E1 -18919.582,E2 -18919.582} C_VEL
LIN {X 0,Y 253.973,Z 488.628,A -85,B 0,C 180,E1 -18920.448,E2 -18920.448} C_VEL
LIN {X 0,Y 255.018,Z 451.114,A -85,B 0,C 180,E1 -18922.11,E2 -18922.11} C_VEL
LIN {X 0,Y 255.337,Z 439.618,A -85,B 0,C 180,E1 -18922.628,E2 -18922.628} C_VEL
LIN {X 0,Y 249.319,Z 418.385,A -85,B 0,C 180,E1 -18923.873,E2 -18923.873} C_VEL
LIN {X 0,Y 249.126,Z 417.517,A -85,B 0,C 180,E1 -18924.202,E2 -18924.202} C_VEL
LIN {X 0,Y 249.04,Z 417.439,A -85,B 0,C 180,E1 -18928.975,E2 -18928.975} C_VEL
LIN {X 0,Y 249.029,Z 417.455,A -85,B 0,C 180,E1 -18932.426,E2 -18932.426} C_VEL
LIN {X 0,Y 249.049,Z 417.463,A -85,B 0,C 180,E1 -18936.342,E2 -18936.342} C_VEL
LIN {X 0,Y 249.048,Z 417.676,A -85,B 0,C 180,E1 -18940.435,E2 -18940.435} C_VEL
LIN {X 0,Y 253.642,Z 429.462,A -85,B 0,C 180,E1 -18944.398,E2 -18944.398} C_VEL
LIN {X 0,Y 257.257,Z 439.71,A -85,B 0,C 180,E1 -18947.529,E2 -18947.529} C_VEL
LIN {X 0,Y 260.27,Z 449.735,A -85,B 0,C 180,E1 -18950.315,E2 -18950.315} C_VEL
LIN {X 0,Y 263.308,Z 462.151,A -85,B 0,C 180,E1 -18953.496,E2 -18953.496} C_VEL
LIN {X 0,Y 264.565,Z 468.951,A -85,B 0,C 180,E1 -18955.1,E2 -18955.1} C_VEL
LIN {X 0,Y 262.311,Z 485.968,A -85,B 0,C 180,E1 -18958.21,E2 -18958.21} C_VEL
LIN {X 0,Y 262.137,Z 488.13,A -85,B 0,C 180,E1 -18958.561,E2 -18958.561} C_VEL
LIN {X 0,Y 266.085,Z 517.161,A -85,B 0,C 180,E1 -18959.984,E2 -18959.984} C_VEL
LIN {X 0,Y 267.23,Z 527.227,A -85,B 0,C 180,E1 -18960.431,E2 -18960.431} C_VEL
LIN {X 0,Y 264.666,Z 601.193,A -85,B 0,C 180,E1 -18962.417,E2 -18962.417} C_VEL
LIN {X 0,Y 263.545,Z 614.369,A -85,B 0,C 180,E1 -18963.042,E2 -18963.042} C_VEL
LIN {X 0,Y 262.029,Z 627.947,A -85,B 0,C 180,E1 -18964.054,E2 -18964.054} C_VEL
LIN {X 0,Y 260.273,Z 639.738,A -85,B 0,C 180,E1 -18965.258,E2 -18965.258} C_VEL
LIN {X 0,Y 258.206,Z 650.965,A -85,B 0,C 180,E1 -18966.755,E2 -18966.755} C_VEL
LIN {X 0,Y 256.183,Z 661.109,A -85,B 0,C 180,E1 -18968.474,E2 -18968.474} C_VEL
LIN {X 0,Y 254.366,Z 669.645,A -85,B 0,C 180,E1 -18970.269,E2 -18970.269} C_VEL
LIN {X 0,Y 252.341,Z 678.451,A -85,B 0,C 180,E1 -18972.579,E2 -18972.579} C_VEL
LIN {X 0,Y 250.547,Z 685.688,A -85,B 0,C 180,E1 -18974.962,E2 -18974.962} C_VEL
LIN {X 0,Y 248.991,Z 692.325,A -85,B 0,C 180,E1 -18977.778,E2 -18977.778} C_VEL
LIN {X 0,Y 248.022,Z 696.683,A -85,B 0,C 180,E1 -18980.211,E2 -18980.211} C_VEL
LIN {X 0,Y 247.598,Z 698.977,A -85,B 0,C 180,E1 -18981.841,E2 -18981.841} C_VEL
LIN {X 0,Y 247.056,Z 701.916,A -85,B 0,C 180,E1 -18984.653,E2 -18984.653} C_VEL
LIN {X 0,Y 246.916,Z 703.272,A -85,B 0,C 180,E1 -18986.737,E2 -18986.737} C_VEL
LIN {X 0,Y 246.88,Z 703.888,A -85,B 0,C 180,E1 -18988.369,E2 -18988.369} C_VEL
LIN {X 0,Y 246.894,Z 704.121,A -85,B 0,C 180,E1 -18990,E2 -18990} C_VEL
LIN {X 0,Y 246.88,Z 703.923,A -85,B 0,C 180,E1 -18991.632,E2 -18991.632} C_VEL
LIN {X 0,Y 246.915,Z 703.331,A -85,B 0,C 180,E1 -18993.264,E2 -18993.264} C_VEL
LIN {X 0,Y 247.023,Z 702.094,A -85,B 0,C 180,E1 -18995.264,E2 -18995.264} C_VEL
LIN {X 0,Y 247.514,Z 699.134,A -85,B 0,C 180,E1 -18998.162,E2 -18998.162} C_VEL
LIN {X 0,Y 248.261,Z 695.556,A -85,B 0,C 180,E1 -19000.604,E2 -19000.604} C_VEL
LIN {X 0,Y 249.327,Z 690.863,A -85,B 0,C 180,E1 -19003.033,E2 -19003.033} C_VEL
LIN {X 0,Y 250.718,Z 684.917,A -85,B 0,C 180,E1 -19005.444,E2 -19005.444} C_VEL
LIN {X 0,Y 252.614,Z 677.518,A -85,B 0,C 180,E1 -19007.821,E2 -19007.821} C_VEL
LIN {X 0,Y 254.513,Z 669.215,A -85,B 0,C 180,E1 -19009.951,E2 -19009.951} C_VEL
LIN {X 0,Y 256.668,Z 658.616,A -85,B 0,C 180,E1 -19012.117,E2 -19012.117} C_VEL
LIN {X 0,Y 258.886,Z 647.88,A -85,B 0,C 180,E1 -19013.817,E2 -19013.817} C_VEL
LIN {X 0,Y 260.982,Z 635.717,A -85,B 0,C 180,E1 -19015.309,E2 -19015.309} C_VEL
LIN {X 0,Y 262.62,Z 623.822,A -85,B 0,C 180,E1 -19016.418,E2 -19016.418} C_VEL
LIN {X 0,Y 263.936,Z 611.482,A -85,B 0,C 180,E1 -19017.237,E2 -19017.237} C_VEL
LIN {X 0,Y 264.942,Z 597.727,A -85,B 0,C 180,E1 -19017.821,E2 -19017.821} C_VEL
LIN {X 0,Y 267.234,Z 525.966,A -85,B 0,C 180,E1 -19019.736,E2 -19019.736} C_VEL
LIN {X 0,Y 263.326,Z 495.838,A -85,B 0,C 180,E1 -19021.159,E2 -19021.159} C_VEL
LIN {X 0,Y 262.197,Z 487.79,A -85,B 0,C 180,E1 -19021.603,E2 -19021.603} C_VEL
LIN {X 0,Y 264.59,Z 468.64,A -85,B 0,C 180,E1 -19025.096,E2 -19025.096} C_VEL
LIN {X 0,Y 262.353,Z 457.635,A -85,B 0,C 180,E1 -19027.791,E2 -19027.791} C_VEL
LIN {X 0,Y 259.58,Z 447.159,A -85,B 0,C 180,E1 -19030.526,E2 -19030.526} C_VEL
LIN {X 0,Y 256.022,Z 435.884,A -85,B 0,C 180,E1 -19033.77,E2 -19033.77} C_VEL
LIN {X 0,Y 252.461,Z 426.339,A -85,B 0,C 180,E1 -19036.774,E2 -19036.774} C_VEL
LIN {X 0,Y 249.045,Z 417.698,A -85,B 0,C 180,E1 -19039.714,E2 -19039.714} C_VEL
LIN {X 0,Y 249.037,Z 417.453,A -85,B 0,C 180,E1 -19042.203,E2 -19042.203} C_VEL
LIN {X 0,Y 249.045,Z 417.452,A -85,B 0,C 180,E1 -19045.639,E2 -19045.639} C_VEL
LIN {X 0,Y 248.997,Z 417.466,A -85,B 0,C 180,E1 -19049.465,E2 -19049.465} C_VEL
LIN {X 0,Y 249.032,Z 417.465,A -85,B 0,C 180,E1 -19053.157,E2 -19053.157} C_VEL
LIN {X 0,Y 249.054,Z 417.441,A -85,B 0,C 180,E1 -19056.73,E2 -19056.73} C_VEL
LIN {X 0,Y 249.039,Z 417.444,A -85,B 0,C 180,E1 -19061.138,E2 -19061.138} C_VEL
LIN {X 0,Y 248.416,Z 417.521,A -85,B 0,C 180,E1 -19062.488,E2 -19062.488} C_VEL
LIN {X 0,Y 245.628,Z 417.887,A -85,B 0,C 180,E1 -19064.691,E2 -19064.691} C_VEL
LIN {X 0,Y 243.248,Z 418.175,A -85,B 0,C 180,E1 -19066.485,E2 -19066.485} C_VEL
LIN {X 0,Y 242.234,Z 418.283,A -85,B 0,C 180,E1 -19067.876,E2 -19067.876} C_VEL
LIN {X 0,Y 242.156,Z 418.29,A -85,B 0,C 180,E1 -19068.346,E2 -19068.346} C_VEL
LIN {X 0,Y 242.384,Z 418.292,A -85,B 0,C 180,E1 -19071.664,E2 -19071.664} C_VEL
LIN {X 0,Y 242.403,Z 418.277,A -85,B 0,C 180,E1 -19073.34,E2 -19073.34} C_VEL
LIN {X 0,Y 242.619,Z 418.261,A -85,B 0,C 180,E1 -19078.34,E2 -19078.34} C_VEL
LIN {X 0,Y 242.618,Z 418.232,A -85,B 0,C 180,E1 -19081.66,E2 -19081.66} C_VEL
LIN {X 0,Y 242.399,Z 418.29,A -85,B 0,C 180,E1 -19086.66,E2 -19086.66} C_VEL
LIN {X 0,Y 242.263,Z 418.275,A -85,B 0,C 180,E1 -19090.024,E2 -19090.024} C_VEL
LIN {X 0,Y 242.108,Z 418.305,A -85,B 0,C 180,E1 -19095.145,E2 -19095.145} C_VEL
LIN {X 0,Y 242.015,Z 418.326,A -85,B 0,C 180,E1 -19098.629,E2 -19098.629} C_VEL
LIN {X 0,Y 241.975,Z 418.319,A -85,B 0,C 180,E1 -19102.184,E2 -19102.184} C_VEL
LIN {X 0,Y 241.988,Z 418.341,A -85,B 0,C 180,E1 -19105.826,E2 -19105.826} C_VEL
LIN {X 0,Y 241.965,Z 418.321,A -85,B 0,C 180,E1 -19109.589,E2 -19109.589} C_VEL
LIN {X 0,Y 241.981,Z 418.326,A -85,B 0,C 180,E1 -19113.493,E2 -19113.493} C_VEL
LIN {X 0,Y 241.982,Z 418.337,A -85,B 0,C 180,E1 -19117.583,E2 -19117.583} C_VEL
LIN {X 0,Y 241.91,Z 418.283,A -85,B 0,C 180,E1 -19121.928,E2 -19121.928} C_VEL
LIN {X 0,Y 241.928,Z 418.571,A -85,B 0,C 180,E1 -19126.34,E2 -19126.34} C_VEL
LIN {X 0,Y 242.358,Z 420.082,A -85,B 0,C 180,E1 -19126.81,E2 -19126.81} C_VEL
LIN {X 0,Y 246.913,Z 427.997,A -85,B 0,C 180,E1 -19128.964,E2 -19128.964} C_VEL
LIN {X 0,Y 249.642,Z 432.99,A -85,B 0,C 180,E1 -19130.212,E2 -19130.212} C_VEL
LIN {X 0,Y 253.763,Z 447.794,A -85,B 0,C 180,E1 -19132.764,E2 -19132.764} C_VEL
LIN {X 0,Y 256.838,Z 459.861,A -85,B 0,C 180,E1 -19134.662,E2 -19134.662} C_VEL
LIN {X 0,Y 256.325,Z 484.853,A -85,B 0,C 180,E1 -19137.446,E2 -19137.446} C_VEL
LIN {X 0,Y 256.312,Z 489.453,A -85,B 0,C 180,E1 -19137.862,E2 -19137.862} C_VEL
LIN {X 0,Y 259.456,Z 519.367,A -85,B 0,C 180,E1 -19139.245,E2 -19139.245} C_VEL
LIN {X 0,Y 260.485,Z 533.539,A -85,B 0,C 180,E1 -19139.822,E2 -19139.822} C_VEL
LIN {X 0,Y 258.166,Z 600.192,A -85,B 0,C 180,E1 -19141.605,E2 -19141.605} C_VEL
LIN {X 0,Y 257.366,Z 613.029,A -85,B 0,C 180,E1 -19142.118,E2 -19142.118} C_VEL
LIN {X 0,Y 256.036,Z 624.924,A -85,B 0,C 180,E1 -19142.848,E2 -19142.848} C_VEL
LIN {X 0,Y 254.6,Z 635.798,A -85,B 0,C 180,E1 -19143.789,E2 -19143.789} C_VEL
LIN {X 0,Y 252.685,Z 647.503,A -85,B 0,C 180,E1 -19145.122,E2 -19145.122} C_VEL
LIN {X 0,Y 250.315,Z 659.133,A -85,B 0,C 180,E1 -19146.854,E2 -19146.854} C_VEL
LIN {X 0,Y 248.081,Z 669.458,A -85,B 0,C 180,E1 -19148.826,E2 -19148.826} C_VEL
LIN {X 0,Y 246.204,Z 677.793,A -85,B 0,C 180,E1 -19150.837,E2 -19150.837} C_VEL
LIN {X 0,Y 244.229,Z 685.914,A -85,B 0,C 180,E1 -19153.276,E2 -19153.276} C_VEL
LIN {X 0,Y 242.545,Z 692.449,A -85,B 0,C 180,E1 -19155.741,E2 -19155.741} C_VEL
LIN {X 0,Y 241.392,Z 697.638,A -85,B 0,C 180,E1 -19158.24,E2 -19158.24} C_VEL
LIN {X 0,Y 240.569,Z 701.644,A -85,B 0,C 180,E1 -19160.753,E2 -19160.753} C_VEL
LIN {X 0,Y 240.091,Z 704.594,A -85,B 0,C 180,E1 -19163.276,E2 -19163.276} C_VEL
LIN {X 0,Y 239.921,Z 706.008,A -85,B 0,C 180,E1 -19164.958,E2 -19164.958} C_VEL
LIN {X 0,Y 239.837,Z 707.007,A -85,B 0,C 180,E1 -19166.64,E2 -19166.64} C_VEL
LIN {X 0,Y 239.847,Z 707.616,A -85,B 0,C 180,E1 -19168.321,E2 -19168.321} C_VEL
LIN {X 0,Y 239.881,Z 707.831,A -85,B 0,C 180,E1 -19170,E2 -19170} C_VEL
LIN {X 0,Y 239.884,Z 707.607,A -85,B 0,C 180,E1 -19171.679,E2 -19171.679} C_VEL
LIN {X 0,Y 239.859,Z 706.99,A -85,B 0,C 180,E1 -19173.359,E2 -19173.359} C_VEL
LIN {X 0,Y 239.944,Z 705.871,A -85,B 0,C 180,E1 -19175.211,E2 -19175.211} C_VEL
LIN {X 0,Y 240.375,Z 702.673,A -85,B 0,C 180,E1 -19178.406,E2 -19178.406} C_VEL
LIN {X 0,Y 241.079,Z 699.013,A -85,B 0,C 180,E1 -19180.923,E2 -19180.923} C_VEL
LIN {X 0,Y 242.103,Z 694.223,A -85,B 0,C 180,E1 -19183.428,E2 -19183.428} C_VEL
LIN {X 0,Y 243.649,Z 688.162,A -85,B 0,C 180,E1 -19185.904,E2 -19185.904} C_VEL
LIN {X 0,Y 245.445,Z 680.603,A -85,B 0,C 180,E1 -19188.359,E2 -19188.359} C_VEL
LIN {X 0,Y 247.426,Z 672.254,A -85,B 0,C 180,E1 -19190.503,E2 -19190.503} C_VEL
LIN {X 0,Y 249.6,Z 662.27,A -85,B 0,C 180,E1 -19192.559,E2 -19192.559} C_VEL
LIN {X 0,Y 251.844,Z 651.469,A -85,B 0,C 180,E1 -19194.306,E2 -19194.306} C_VEL
LIN {X 0,Y 254.043,Z 639.16,A -85,B 0,C 180,E1 -19195.831,E2 -19195.831} C_VEL
LIN {X 0,Y 254.435,Z 636.853,A -85,B 0,C 180,E1 -19196.118,E2 -19196.118} C_VEL
LIN {X 0,Y 259.308,Z 627.472,A -85,B 0,C 180,E1 -19198.314,E2 -19198.314} C_VEL
LIN {X 0,Y 264.674,Z 616.655,A -85,B 0,C 180,E1 -19200.299,E2 -19200.299} C_VEL
LIN {X 0,Y 270.113,Z 604.699,A -85,B 0,C 180,E1 -19202.014,E2 -19202.014} C_VEL
LIN {X 0,Y 275.386,Z 591.557,A -85,B 0,C 180,E1 -19203.496,E2 -19203.496} C_VEL
LIN {X 0,Y 279.962,Z 578.698,A -85,B 0,C 180,E1 -19204.608,E2 -19204.608} C_VEL
LIN {X 0,Y 284.322,Z 563.794,A -85,B 0,C 180,E1 -19205.622,E2 -19205.622} C_VEL
LIN {X 0,Y 287.932,Z 547.761,A -85,B 0,C 180,E1 -19206.455,E2 -19206.455} C_VEL
LIN {X 0,Y 289.693,Z 536.957,A -85,B 0,C 180,E1 -19207.01,E2 -19207.01} C_VEL
LIN {X 0,Y 290.963,Z 526.523,A -85,B 0,C 180,E1 -19207.769,E2 -19207.769} C_VEL
LIN {X 0,Y 292.262,Z 513.132,A -85,B 0,C 180,E1 -19209.035,E2 -19209.035} C_VEL
LIN {X 0,Y 293.34,Z 500.595,A -85,B 0,C 180,E1 -19210.538,E2 -19210.538} C_VEL
LIN {X 0,Y 293.415,Z 499.032,A -85,B 0,C 180,E1 -19210.799,E2 -19210.799} C_VEL
LIN {X 0,Y 293.026,Z 495.403,A -85,B 0,C 180,E1 -19211.968,E2 -19211.968} C_VEL
LIN {X 0,Y 292.501,Z 490.417,A -85,B 0,C 180,E1 -19214.421,E2 -19214.421} C_VEL
LIN {X 0,Y 292.639,Z 487.902,A -85,B 0,C 180,E1 -19216.352,E2 -19216.352} C_VEL
LIN {X 0,Y 293.405,Z 486.448,A -85,B 0,C 180,E1 -19218.515,E2 -19218.515} C_VEL
LIN {X 0,Y 294.899,Z 486.36,A -85,B 0,C 180,E1 -19220.746,E2 -19220.746} C_VEL
LIN {X 0,Y 296.399,Z 487.209,A -85,B 0,C 180,E1 -19222.321,E2 -19222.321} C_VEL
LIN {X 0,Y 297.558,Z 488.269,A -85,B 0,C 180,E1 -19223.347,E2 -19223.347} C_VEL
LIN {X 0,Y 292.197,Z 517.971,A -85,B 0,C 180,E1 -19224.9,E2 -19224.9} C_VEL
LIN {X 0,Y 289.729,Z 531.916,A -85,B 0,C 180,E1 -19225.879,E2 -19225.879} C_VEL
LIN {X 0,Y 286.718,Z 544.133,A -85,B 0,C 180,E1 -19226.949,E2 -19226.949} C_VEL
LIN {X 0,Y 282.622,Z 557.527,A -85,B 0,C 180,E1 -19228.519,E2 -19228.519} C_VEL
LIN {X 0,Y 278.532,Z 568.383,A -85,B 0,C 180,E1 -19230.11,E2 -19230.11} C_VEL
LIN {X 0,Y 274.601,Z 577.268,A -85,B 0,C 180,E1 -19231.74,E2 -19231.74} C_VEL
LIN {X 0,Y 270.893,Z 584.736,A -85,B 0,C 180,E1 -19233.415,E2 -19233.415} C_VEL
LIN {X 0,Y 266.702,Z 592.045,A -85,B 0,C 180,E1 -19235.478,E2 -19235.478} C_VEL
LIN {X 0,Y 262.169,Z 598.917,A -85,B 0,C 180,E1 -19237.957,E2 -19237.957} C_VEL
LIN {X 0,Y 258.54,Z 603.456,A -85,B 0,C 180,E1 -19240.136,E2 -19240.136} C_VEL
LIN {X 0,Y 255.326,Z 606.889,A -85,B 0,C 180,E1 -19242.375,E2 -19242.375} C_VEL
LIN {X 0,Y 253.304,Z 608.639,A -85,B 0,C 180,E1 -19243.892,E2 -19243.892} C_VEL
LIN {X 0,Y 251.559,Z 609.924,A -85,B 0,C 180,E1 -19245.437,E2 -19245.437} C_VEL
LIN {X 0,Y 249.878,Z 610.78,A -85,B 0,C 180,E1 -19246.997,E2 -19246.997} C_VEL
LIN {X 0,Y 246.997,Z 611.274,A -85,B 0,C 180,E1 -19250.17,E2 -19250.17} C_VEL
LIN {X 0,Y 245.819,Z 610.908,A -85,B 0,C 180,E1 -19251.781,E2 -19251.781} C_VEL
LIN {X 0,Y 244.991,Z 610.062,A -85,B 0,C 180,E1 -19253.411,E2 -19253.411} C_VEL
LIN {X 0,Y 244.253,Z 608.825,A -85,B 0,C 180,E1 -19255.048,E2 -19255.048} C_VEL
LIN {X 0,Y 243.163,Z 606.211,A -85,B 0,C 180,E1 -19257.515,E2 -19257.515} C_VEL
LIN {X 0,Y 242.322,Z 602.588,A -85,B 0,C 180,E1 -19260,E2 -19260} C_VEL
LIN {X 0,Y 242.055,Z 597.873,A -85,B 0,C 180,E1 -19262.496,E2 -19262.496} C_VEL
LIN {X 0,Y 242.031,Z 590.877,A -85,B 0,C 180,E1 -19265.415,E2 -19265.415} C_VEL
LIN {X 0,Y 242.37,Z 583.31,A -85,B 0,C 180,E1 -19267.917,E2 -19267.917} C_VEL
LIN {X 0,Y 242.845,Z 574.215,A -85,B 0,C 180,E1 -19270.378,E2 -19270.378} C_VEL
LIN {X 0,Y 243.464,Z 563.574,A -85,B 0,C 180,E1 -19272.716,E2 -19272.716} C_VEL
LIN {X 0,Y 244.202,Z 551.929,A -85,B 0,C 180,E1 -19274.798,E2 -19274.798} C_VEL
LIN {X 0,Y 244.997,Z 538.838,A -85,B 0,C 180,E1 -19276.67,E2 -19276.67} C_VEL
LIN {X 0,Y 245.829,Z 524.913,A -85,B 0,C 180,E1 -19278.222,E2 -19278.222} C_VEL
LIN {X 0,Y 246.34,Z 510.856,A -85,B 0,C 180,E1 -19279.408,E2 -19279.408} C_VEL
LIN {X 0,Y 246.703,Z 496.36,A -85,B 0,C 180,E1 -19280.262,E2 -19280.262} C_VEL
LIN {X 0,Y 248.165,Z 446.841,A -85,B 0,C 180,E1 -19282.538,E2 -19282.538} C_VEL
LIN {X 0,Y 248.311,Z 440.777,A -85,B 0,C 180,E1 -19282.819,E2 -19282.819} C_VEL
LIN {X 0,Y 242.245,Z 419.231,A -85,B 0,C 180,E1 -19284.127,E2 -19284.127} C_VEL
LIN {X 0,Y 242.098,Z 418.407,A -85,B 0,C 180,E1 -19284.436,E2 -19284.436} C_VEL
LIN {X 0,Y 241.971,Z 418.322,A -85,B 0,C 180,E1 -19289.588,E2 -19289.588} C_VEL
LIN {X 0,Y 241.981,Z 418.323,A -85,B 0,C 180,E1 -19293.493,E2 -19293.493} C_VEL
LIN {X 0,Y 241.99,Z 418.328,A -85,B 0,C 180,E1 -19297.582,E2 -19297.582} C_VEL
LIN {X 0,Y 242.048,Z 418.638,A -85,B 0,C 180,E1 -19298.996,E2 -19298.996} C_VEL
LIN {X 0,Y 246.725,Z 430.328,A -85,B 0,C 180,E1 -19303.129,E2 -19303.129} C_VEL
LIN {X 0,Y 250.829,Z 441.734,A -85,B 0,C 180,E1 -19306.761,E2 -19306.761} C_VEL
LIN {X 0,Y 254.027,Z 452.549,A -85,B 0,C 180,E1 -19309.866,E2 -19309.866} C_VEL
LIN {X 0,Y 256.908,Z 464.534,A -85,B 0,C 180,E1 -19312.999,E2 -19312.999} C_VEL
LIN {X 0,Y 258.159,Z 471.398,A -85,B 0,C 180,E1 -19314.656,E2 -19314.656} C_VEL
LIN {X 0,Y 256.115,Z 485.966,A -85,B 0,C 180,E1 -19317.347,E2 -19317.347} C_VEL
LIN {X 0,Y 255.947,Z 488.428,A -85,B 0,C 180,E1 -19317.727,E2 -19317.727} C_VEL
LIN {X 0,Y 259.868,Z 517.276,A -85,B 0,C 180,E1 -19319.193,E2 -19319.193} C_VEL
LIN {X 0,Y 261.056,Z 528.543,A -85,B 0,C 180,E1 -19319.702,E2 -19319.702} C_VEL
LIN {X 0,Y 258.413,Z 601.189,A -85,B 0,C 180,E1 -19321.69,E2 -19321.69} C_VEL
LIN {X 0,Y 257.235,Z 614.394,A -85,B 0,C 180,E1 -19322.325,E2 -19322.325} C_VEL
LIN {X 0,Y 255.654,Z 627.984,A -85,B 0,C 180,E1 -19323.357,E2 -19323.357} C_VEL
LIN {X 0,Y 253.841,Z 639.781,A -85,B 0,C 180,E1 -19324.587,E2 -19324.587} C_VEL
LIN {X 0,Y 251.713,Z 651.012,A -85,B 0,C 180,E1 -19326.118,E2 -19326.118} C_VEL
LIN {X 0,Y 249.567,Z 661.159,A -85,B 0,C 180,E1 -19327.874,E2 -19327.874} C_VEL
LIN {X 0,Y 247.345,Z 671.118,A -85,B 0,C 180,E1 -19330.064,E2 -19330.064} C_VEL
LIN {X 0,Y 245.212,Z 679.832,A -85,B 0,C 180,E1 -19332.486,E2 -19332.486} C_VEL
LIN {X 0,Y 243.373,Z 686.824,A -85,B 0,C 180,E1 -19334.936,E2 -19334.936} C_VEL
LIN {X 0,Y 242.039,Z 692.379,A -85,B 0,C 180,E1 -19337.422,E2 -19337.422} C_VEL
LIN {X 0,Y 241.004,Z 696.738,A -85,B 0,C 180,E1 -19339.923,E2 -19339.923} C_VEL
LIN {X 0,Y 240.549,Z 699.031,A -85,B 0,C 180,E1 -19341.6,E2 -19341.6} C_VEL
LIN {X 0,Y 239.945,Z 702.211,A -85,B 0,C 180,E1 -19344.789,E2 -19344.789} C_VEL
LIN {X 0,Y 239.825,Z 703.326,A -85,B 0,C 180,E1 -19346.64,E2 -19346.64} C_VEL
LIN {X 0,Y 239.796,Z 703.942,A -85,B 0,C 180,E1 -19348.321,E2 -19348.321} C_VEL
LIN {X 0,Y 239.806,Z 704.175,A -85,B 0,C 180,E1 -19350,E2 -19350} C_VEL
LIN {X 0,Y 239.796,Z 703.977,A -85,B 0,C 180,E1 -19351.68,E2 -19351.68} C_VEL
LIN {X 0,Y 239.823,Z 703.385,A -85,B 0,C 180,E1 -19353.36,E2 -19353.36} C_VEL
LIN {X 0,Y 239.92,Z 702.341,A -85,B 0,C 180,E1 -19355.146,E2 -19355.146} C_VEL
LIN {X 0,Y 240.143,Z 701.029,A -85,B 0,C 180,E1 -19356.723,E2 -19356.723} C_VEL
LIN {X 0,Y 240.718,Z 698.133,A -85,B 0,C 180,E1 -19359.241,E2 -19359.241} C_VEL
LIN {X 0,Y 241.602,Z 694.198,A -85,B 0,C 180,E1 -19361.749,E2 -19361.749} C_VEL
LIN {X 0,Y 242.838,Z 689.099,A -85,B 0,C 180,E1 -19364.241,E2 -19364.241} C_VEL
LIN {X 0,Y 244.501,Z 682.672,A -85,B 0,C 180,E1 -19366.705,E2 -19366.705} C_VEL
LIN {X 0,Y 246.578,Z 674.686,A -85,B 0,C 180,E1 -19369.134,E2 -19369.134} C_VEL
LIN {X 0,Y 248.467,Z 666.411,A -85,B 0,C 180,E1 -19371.167,E2 -19371.167} C_VEL
LIN {X 0,Y 250.589,Z 656.464,A -85,B 0,C 180,E1 -19373.119,E2 -19373.119} C_VEL
LIN {X 0,Y 252.951,Z 645.154,A -85,B 0,C 180,E1 -19374.85,E2 -19374.85} C_VEL
LIN {X 0,Y 254.861,Z 634.015,A -85,B 0,C 180,E1 -19376.182,E2 -19376.182} C_VEL
LIN {X 0,Y 256.545,Z 621.386,A -85,B 0,C 180,E1 -19377.314,E2 -19377.314} C_VEL
LIN {X 0,Y 257.916,Z 608.938,A -85,B 0,C 180,E1 -19378.093,E2 -19378.093} C_VEL
LIN {X 0,Y 258.778,Z 596.121,A -85,B 0,C 180,E1 -19378.599,E2 -19378.599} C_VEL
LIN {X 0,Y 261.023,Z 526.328,A -85,B 0,C 180,E1 -19380.503,E2 -19380.503} C_VEL
LIN {X 0,Y 257.259,Z 496.953,A -85,B 0,C 180,E1 -19381.941,E2 -19381.941} C_VEL
LIN {X 0,Y 255.955,Z 487.778,A -85,B 0,C 180,E1 -19382.467,E2 -19382.467} C_VEL
LIN {X 0,Y 258.212,Z 471.432,A -85,B 0,C 180,E1 -19385.479,E2 -19385.479} C_VEL
LIN {X 0,Y 257.153,Z 465.277,A -85,B 0,C 180,E1 -19386.961,E2 -19386.961} C_VEL
LIN {X 0,Y 254.598,Z 454.373,A -85,B 0,C 180,E1 -19389.794,E2 -19389.794} C_VEL
LIN {X 0,Y 250.95,Z 442.222,A -85,B 0,C 180,E1 -19393.269,E2 -19393.269} C_VEL
LIN {X 0,Y 247.508,Z 432.394,A -85,B 0,C 180,E1 -19396.379,E2 -19396.379} C_VEL
LIN {X 0,Y 243.895,Z 423.517,A -85,B 0,C 180,E1 -19399.385,E2 -19399.385} C_VEL
LIN {X 0,Y 242,Z 418.55,A -85,B 0,C 180,E1 -19401.243,E2 -19401.243} C_VEL
LIN {X 0,Y 241.981,Z 418.344,A -85,B 0,C 180,E1 -19404.488,E2 -19404.488} C_VEL
LIN {X 0,Y 241.952,Z 418.346,A -85,B 0,C 180,E1 -19408.476,E2 -19408.476} C_VEL
LIN {X 0,Y 241.963,Z 418.333,A -85,B 0,C 180,E1 -19412.307,E2 -19412.307} C_VEL
LIN {X 0,Y 242.026,Z 418.316,A -85,B 0,C 180,E1 -19416.012,E2 -19416.012} C_VEL
LIN {X 0,Y 241.988,Z 418.342,A -85,B 0,C 180,E1 -19419.603,E2 -19419.603} C_VEL
LIN {X 0,Y 242.108,Z 418.306,A -85,B 0,C 180,E1 -19423.324,E2 -19423.324} C_VEL
LIN {X 0,Y 242.156,Z 418.29,A -85,B 0,C 180,E1 -19428.346,E2 -19428.346} C_VEL
LIN {X 0,Y 241.496,Z 418.381,A -85,B 0,C 180,E1 -19429.738,E2 -19429.738} C_VEL
LIN {X 0,Y 238.646,Z 418.759,A -85,B 0,C 180,E1 -19432.009,E2 -19432.009} C_VEL
LIN {X 0,Y 236.248,Z 419.039,A -85,B 0,C 180,E1 -19433.859,E2 -19433.859} C_VEL
LIN {X 0,Y 235.261,Z 419.147,A -85,B 0,C 180,E1 -19435.295,E2 -19435.295} C_VEL
LIN {X 0,Y 235.203,Z 419.154,A -85,B 0,C 180,E1 -19435.781,E2 -19435.781} C_VEL
LIN {X 0,Y 235.578,Z 419.137,A -85,B 0,C 180,E1 -19438.29,E2 -19438.29} C_VEL
LIN {X 0,Y 235.577,Z 419.108,A -85,B 0,C 180,E1 -19441.709,E2 -19441.709} C_VEL
LIN {X 0,Y 235.35,Z 419.166,A -85,B 0,C 180,E1 -19446.86,E2 -19446.86} C_VEL
LIN {X 0,Y 235.187,Z 419.157,A -85,B 0,C 180,E1 -19450.329,E2 -19450.329} C_VEL
LIN {X 0,Y 235.045,Z 419.179,A -85,B 0,C 180,E1 -19455.611,E2 -19455.611} C_VEL
LIN {X 0,Y 234.958,Z 419.215,A -85,B 0,C 180,E1 -19459.21,E2 -19459.21} C_VEL
LIN {X 0,Y 234.91,Z 419.195,A -85,B 0,C 180,E1 -19462.888,E2 -19462.888} C_VEL
LIN {X 0,Y 234.924,Z 419.221,A -85,B 0,C 180,E1 -19466.663,E2 -19466.663} C_VEL
LIN {X 0,Y 234.897,Z 419.21,A -85,B 0,C 180,E1 -19470.573,E2 -19470.573} C_VEL
LIN {X 0,Y 234.926,Z 419.201,A -85,B 0,C 180,E1 -19474.639,E2 -19474.639} C_VEL
LIN {X 0,Y 234.913,Z 419.178,A -85,B 0,C 180,E1 -19478.935,E2 -19478.935} C_VEL
LIN {X 0,Y 234.858,Z 419.178,A -85,B 0,C 180,E1 -19483.493,E2 -19483.493} C_VEL
LIN {X 0,Y 234.901,Z 419.474,A -85,B 0,C 180,E1 -19484.608,E2 -19484.608} C_VEL
LIN {X 0,Y 235.539,Z 421.5,A -85,B 0,C 180,E1 -19485.243,E2 -19485.243} C_VEL
LIN {X 0,Y 236.89,Z 423.352,A -85,B 0,C 180,E1 -19485.876,E2 -19485.876} C_VEL
LIN {X 0,Y 244.024,Z 436.287,A -85,B 0,C 180,E1 -19489.376,E2 -19489.376} C_VEL
LIN {X 0,Y 244.959,Z 438.68,A -85,B 0,C 180,E1 -19489.898,E2 -19489.898} C_VEL
LIN {X 0,Y 248.902,Z 454.165,A -85,B 0,C 180,E1 -19492.603,E2 -19492.603} C_VEL
LIN {X 0,Y 250.977,Z 462.57,A -85,B 0,C 180,E1 -19493.981,E2 -19493.981} C_VEL
LIN {X 0,Y 250.176,Z 488.754,A -85,B 0,C 180,E1 -19496.947,E2 -19496.947} C_VEL
LIN {X 0,Y 252.969,Z 516.354,A -85,B 0,C 180,E1 -19498.265,E2 -19498.265} C_VEL
LIN {X 0,Y 254.339,Z 534.828,A -85,B 0,C 180,E1 -19499.052,E2 -19499.052} C_VEL
LIN {X 0,Y 251.966,Z 600.255,A -85,B 0,C 180,E1 -19500.84,E2 -19500.84} C_VEL
LIN {X 0,Y 251.025,Z 613.916,A -85,B 0,C 180,E1 -19501.407,E2 -19501.407} C_VEL
LIN {X 0,Y 249.598,Z 626.175,A -85,B 0,C 180,E1 -19502.202,E2 -19502.202} C_VEL
LIN {X 0,Y 247.97,Z 637.676,A -85,B 0,C 180,E1 -19503.26,E2 -19503.26} C_VEL
LIN {X 0,Y 245.982,Z 648.875,A -85,B 0,C 180,E1 -19504.623,E2 -19504.623} C_VEL
LIN {X 0,Y 243.547,Z 660.252,A -85,B 0,C 180,E1 -19506.397,E2 -19506.397} C_VEL
LIN {X 0,Y 241.45,Z 669.413,A -85,B 0,C 180,E1 -19508.215,E2 -19508.215} C_VEL
LIN {X 0,Y 239.413,Z 678.076,A -85,B 0,C 180,E1 -19510.371,E2 -19510.371} C_VEL
LIN {X 0,Y 237.418,Z 685.865,A -85,B 0,C 180,E1 -19512.781,E2 -19512.781} C_VEL
LIN {X 0,Y 235.645,Z 692.398,A -85,B 0,C 180,E1 -19515.314,E2 -19515.314} C_VEL
LIN {X 0,Y 234.414,Z 697.586,A -85,B 0,C 180,E1 -19517.885,E2 -19517.885} C_VEL
LIN {X 0,Y 233.53,Z 701.591,A -85,B 0,C 180,E1 -19520.472,E2 -19520.472} C_VEL
LIN {X 0,Y 233.017,Z 704.541,A -85,B 0,C 180,E1 -19523.07,E2 -19523.07} C_VEL
LIN {X 0,Y 232.832,Z 706.042,A -85,B 0,C 180,E1 -19524.939,E2 -19524.939} C_VEL
LIN {X 0,Y 232.761,Z 707.563,A -85,B 0,C 180,E1 -19528.269,E2 -19528.269} C_VEL
LIN {X 0,Y 232.792,Z 707.777,A -85,B 0,C 180,E1 -19530,E2 -19530} C_VEL
LIN {X 0,Y 232.796,Z 707.552,A -85,B 0,C 180,E1 -19531.73,E2 -19531.73} C_VEL
LIN {X 0,Y 232.844,Z 705.931,A -85,B 0,C 180,E1 -19535.195,E2 -19535.195} C_VEL
LIN {X 0,Y 233.02,Z 704.504,A -85,B 0,C 180,E1 -19536.929,E2 -19536.929} C_VEL
LIN {X 0,Y 233.534,Z 701.539,A -85,B 0,C 180,E1 -19539.527,E2 -19539.527} C_VEL
LIN {X 0,Y 234.415,Z 697.515,A -85,B 0,C 180,E1 -19542.114,E2 -19542.114} C_VEL
LIN {X 0,Y 235.891,Z 691.309,A -85,B 0,C 180,E1 -19545.111,E2 -19545.111} C_VEL
LIN {X 0,Y 237.76,Z 684.539,A -85,B 0,C 180,E1 -19547.637,E2 -19547.637} C_VEL
LIN {X 0,Y 239.698,Z 676.833,A -85,B 0,C 180,E1 -19549.934,E2 -19549.934} C_VEL
LIN {X 0,Y 241.871,Z 667.306,A -85,B 0,C 180,E1 -19552.194,E2 -19552.194} C_VEL
LIN {X 0,Y 244.34,Z 656.547,A -85,B 0,C 180,E1 -19554.197,E2 -19554.197} C_VEL
LIN {X 0,Y 246.52,Z 645.653,A -85,B 0,C 180,E1 -19555.77,E2 -19555.77} C_VEL
LIN {X 0,Y 247.805,Z 638.463,A -85,B 0,C 180,E1 -19556.645,E2 -19556.645} C_VEL
LIN {X 0,Y 253.168,Z 629.034,A -85,B 0,C 180,E1 -19559.065,E2 -19559.065} C_VEL
LIN {X 0,Y 258.679,Z 618.906,A -85,B 0,C 180,E1 -19561.078,E2 -19561.078} C_VEL
LIN {X 0,Y 264.774,Z 606.753,A -85,B 0,C 180,E1 -19562.966,E2 -19562.966} C_VEL
LIN {X 0,Y 270.804,Z 593.137,A -85,B 0,C 180,E1 -19564.591,E2 -19564.591} C_VEL
LIN {X 0,Y 275.49,Z 581.139,A -85,B 0,C 180,E1 -19565.701,E2 -19565.701} C_VEL
LIN {X 0,Y 280.697,Z 565.366,A -85,B 0,C 180,E1 -19566.823,E2 -19566.823} C_VEL
LIN {X 0,Y 284.814,Z 549.282,A -85,B 0,C 180,E1 -19567.697,E2 -19567.697} C_VEL
LIN {X 0,Y 286.769,Z 538.657,A -85,B 0,C 180,E1 -19568.248,E2 -19568.248} C_VEL
LIN {X 0,Y 288.321,Z 527.476,A -85,B 0,C 180,E1 -19569.085,E2 -19569.085} C_VEL
LIN {X 0,Y 289.877,Z 514.315,A -85,B 0,C 180,E1 -19570.393,E2 -19570.393} C_VEL
LIN {X 0,Y 291.034,Z 504.151,A -85,B 0,C 180,E1 -19571.672,E2 -19571.672} C_VEL
LIN {X 0,Y 290.846,Z 501.159,A -85,B 0,C 180,E1 -19572.689,E2 -19572.689} C_VEL
LIN {X 0,Y 290.63,Z 496.641,A -85,B 0,C 180,E1 -19575.035,E2 -19575.035} C_VEL
LIN {X 0,Y 290.943,Z 494.434,A -85,B 0,C 180,E1 -19576.888,E2 -19576.888} C_VEL
LIN {X 0,Y 291.922,Z 493.162,A -85,B 0,C 180,E1 -19579.122,E2 -19579.122} C_VEL
LIN {X 0,Y 293.797,Z 493.537,A -85,B 0,C 180,E1 -19581.541,E2 -19581.541} C_VEL
LIN {X 0,Y 294.501,Z 494.108,A -85,B 0,C 180,E1 -19582.272,E2 -19582.272} C_VEL
LIN {X 0,Y 289.309,Z 521.312,A -85,B 0,C 180,E1 -19583.746,E2 -19583.746} C_VEL
LIN {X 0,Y 286.303,Z 535.93,A -85,B 0,C 180,E1 -19584.823,E2 -19584.823} C_VEL
LIN {X 0,Y 282.781,Z 548.528,A -85,B 0,C 180,E1 -19586,E2 -19586} C_VEL
LIN {X 0,Y 278.869,Z 560.123,A -85,B 0,C 180,E1 -19587.415,E2 -19587.415} C_VEL
LIN {X 0,Y 274.079,Z 571.557,A -85,B 0,C 180,E1 -19589.146,E2 -19589.146} C_VEL
LIN {X 0,Y 269.124,Z 581.69,A -85,B 0,C 180,E1 -19591.111,E2 -19591.111} C_VEL
LIN {X 0,Y 264.489,Z 589.779,A -85,B 0,C 180,E1 -19593.146,E2 -19593.146} C_VEL
LIN {X 0,Y 260.15,Z 596.429,A -85,B 0,C 180,E1 -19595.245,E2 -19595.245} C_VEL
LIN {X 0,Y 256.06,Z 601.737,A -85,B 0,C 180,E1 -19597.403,E2 -19597.403} C_VEL
LIN {X 0,Y 252.292,Z 605.967,A -85,B 0,C 180,E1 -19599.622,E2 -19599.622} C_VEL
LIN {X 0,Y 248.882,Z 609.086,A -85,B 0,C 180,E1 -19601.903,E2 -19601.903} C_VEL
LIN {X 0,Y 246.781,Z 610.614,A -85,B 0,C 180,E1 -19603.454,E2 -19603.454} C_VEL
LIN {X 0,Y 243.164,Z 612.396,A -85,B 0,C 180,E1 -19606.631,E2 -19606.631} C_VEL
LIN {X 0,Y 241.549,Z 612.693,A -85,B 0,C 180,E1 -19608.248,E2 -19608.248} C_VEL
LIN {X 0,Y 240.139,Z 612.541,A -85,B 0,C 180,E1 -19609.887,E2 -19609.887} C_VEL
LIN {X 0,Y 238.893,Z 611.978,A -85,B 0,C 180,E1 -19611.541,E2 -19611.541} C_VEL
LIN {X 0,Y 238.012,Z 610.991,A -85,B 0,C 180,E1 -19613.217,E2 -19613.217} C_VEL
LIN {X 0,Y 237.234,Z 609.61,A -85,B 0,C 180,E1 -19614.901,E2 -19614.901} C_VEL
LIN {X 0,Y 236.095,Z 606.746,A -85,B 0,C 180,E1 -19617.441,E2 -19617.441} C_VEL
LIN {X 0,Y 235.229,Z 602.877,A -85,B 0,C 180,E1 -19620,E2 -19620} C_VEL
LIN {X 0,Y 234.962,Z 597.868,A -85,B 0,C 180,E1 -19622.572,E2 -19622.572} C_VEL
LIN {X 0,Y 234.944,Z 590.458,A -85,B 0,C 180,E1 -19625.579,E2 -19625.579} C_VEL
LIN {X 0,Y 235.353,Z 581.913,A -85,B 0,C 180,E1 -19628.352,E2 -19628.352} C_VEL
LIN {X 0,Y 235.855,Z 572.916,A -85,B 0,C 180,E1 -19630.733,E2 -19630.733} C_VEL
LIN {X 0,Y 236.507,Z 561.96,A -85,B 0,C 180,E1 -19633.096,E2 -19633.096} C_VEL
LIN {X 0,Y 237.241,Z 549.593,A -85,B 0,C 180,E1 -19635.243,E2 -19635.243} C_VEL
LIN {X 0,Y 237.999,Z 537.296,A -85,B 0,C 180,E1 -19636.954,E2 -19636.954} C_VEL
LIN {X 0,Y 238.792,Z 523.753,A -85,B 0,C 180,E1 -19638.445,E2 -19638.445} C_VEL
LIN {X 0,Y 239.301,Z 508.384,A -85,B 0,C 180,E1 -19639.698,E2 -19639.698} C_VEL
LIN {X 0,Y 239.737,Z 492.125,A -85,B 0,C 180,E1 -19640.597,E2 -19640.597} C_VEL
LIN {X 0,Y 241.179,Z 446.424,A -85,B 0,C 180,E1 -19642.806,E2 -19642.806} C_VEL
LIN {X 0,Y 241.126,Z 441.414,A -85,B 0,C 180,E1 -19643.053,E2 -19643.053} C_VEL
LIN {X 0,Y 235.204,Z 420.063,A -85,B 0,C 180,E1 -19644.373,E2 -19644.373} C_VEL
LIN {X 0,Y 235.044,Z 419.298,A -85,B 0,C 180,E1 -19644.667,E2 -19644.667} C_VEL
LIN {X 0,Y 234.925,Z 419.201,A -85,B 0,C 180,E1 -19649.823,E2 -19649.823} C_VEL
LIN {X 0,Y 234.942,Z 419.201,A -85,B 0,C 180,E1 -19653.114,E2 -19653.114} C_VEL
LIN {X 0,Y 234.968,Z 419.415,A -85,B 0,C 180,E1 -19657.279,E2 -19657.279} C_VEL
LIN {X 0,Y 237.788,Z 426.221,A -85,B 0,C 180,E1 -19659.949,E2 -19659.949} C_VEL
LIN {X 0,Y 241.832,Z 436.518,A -85,B 0,C 180,E1 -19663.59,E2 -19663.59} C_VEL
LIN {X 0,Y 244.929,Z 445.494,A -85,B 0,C 180,E1 -19666.476,E2 -19666.476} C_VEL
LIN {X 0,Y 247.926,Z 455.791,A -85,B 0,C 180,E1 -19669.49,E2 -19669.49} C_VEL
LIN {X 0,Y 251.111,Z 469.262,A -85,B 0,C 180,E1 -19673.071,E2 -19673.071} C_VEL
LIN {X 0,Y 251.782,Z 473.565,A -85,B 0,C 180,E1 -19674.114,E2 -19674.114} C_VEL
LIN {X 0,Y 249.843,Z 487.066,A -85,B 0,C 180,E1 -19676.638,E2 -19676.638} C_VEL
LIN {X 0,Y 249.81,Z 488.657,A -85,B 0,C 180,E1 -19676.846,E2 -19676.846} C_VEL
LIN {X 0,Y 253.332,Z 514.489,A -85,B 0,C 180,E1 -19678.217,E2 -19678.217} C_VEL
LIN {X 0,Y 254.921,Z 529.092,A -85,B 0,C 180,E1 -19678.912,E2 -19678.912} C_VEL
LIN {X 0,Y 252.203,Z 601.185,A -85,B 0,C 180,E1 -19680.927,E2 -19680.927} C_VEL
LIN {X 0,Y 250.976,Z 614.42,A -85,B 0,C 180,E1 -19681.573,E2 -19681.573} C_VEL
LIN {X 0,Y 249.325,Z 628.021,A -85,B 0,C 180,E1 -19682.625,E2 -19682.625} C_VEL
LIN {X 0,Y 247.444,Z 639.825,A -85,B 0,C 180,E1 -19683.881,E2 -19683.881} C_VEL
LIN {X 0,Y 245.237,Z 651.059,A -85,B 0,C 180,E1 -19685.447,E2 -19685.447} C_VEL
LIN {X 0,Y 242.983,Z 661.209,A -85,B 0,C 180,E1 -19687.241,E2 -19687.241} C_VEL
LIN {X 0,Y 241.13,Z 669.391,A -85,B 0,C 180,E1 -19689.045,E2 -19689.045} C_VEL
LIN {X 0,Y 239.168,Z 677.215,A -85,B 0,C 180,E1 -19691.141,E2 -19691.141} C_VEL
LIN {X 0,Y 237.102,Z 684.7,A -85,B 0,C 180,E1 -19693.645,E2 -19693.645} C_VEL
LIN {X 0,Y 235.554,Z 690.704,A -85,B 0,C 180,E1 -19696.191,E2 -19696.191} C_VEL
LIN {X 0,Y 234.339,Z 695.453,A -85,B 0,C 180,E1 -19698.759,E2 -19698.759} C_VEL
LIN {X 0,Y 233.51,Z 699.086,A -85,B 0,C 180,E1 -19701.345,E2 -19701.345} C_VEL
LIN {X 0,Y 233.129,Z 700.956,A -85,B 0,C 180,E1 -19703.074,E2 -19703.074} C_VEL
LIN {X 0,Y 232.832,Z 702.469,A -85,B 0,C 180,E1 -19704.942,E2 -19704.942} C_VEL
LIN {X 0,Y 232.695,Z 703.996,A -85,B 0,C 180,E1 -19708.269,E2 -19708.269} C_VEL
LIN {X 0,Y 232.721,Z 704.229,A -85,B 0,C 180,E1 -19710,E2 -19710} C_VEL
LIN {X 0,Y 232.695,Z 704.031,A -85,B 0,C 180,E1 -19711.731,E2 -19711.731} C_VEL
LIN {X 0,Y 232.836,Z 702.543,A -85,B 0,C 180,E1 -19715.069,E2 -19715.069} C_VEL
LIN {X 0,Y 233.082,Z 701.083,A -85,B 0,C 180,E1 -19716.928,E2 -19716.928} C_VEL
LIN {X 0,Y 233.714,Z 698.185,A -85,B 0,C 180,E1 -19719.52,E2 -19719.52} C_VEL
LIN {X 0,Y 234.636,Z 694.25,A -85,B 0,C 180,E1 -19722.103,E2 -19722.103} C_VEL
LIN {X 0,Y 235.927,Z 689.149,A -85,B 0,C 180,E1 -19724.668,E2 -19724.668} C_VEL
LIN {X 0,Y 237.697,Z 682.721,A -85,B 0,C 180,E1 -19727.198,E2 -19727.198} C_VEL
LIN {X 0,Y 239.841,Z 674.734,A -85,B 0,C 180,E1 -19729.693,E2 -19729.693} C_VEL
LIN {X 0,Y 241.876,Z 666.259,A -85,B 0,C 180,E1 -19731.823,E2 -19731.823} C_VEL
LIN {X 0,Y 244.075,Z 656.505,A -85,B 0,C 180,E1 -19733.774,E2 -19733.774} C_VEL
LIN {X 0,Y 246.53,Z 645.19,A -85,B 0,C 180,E1 -19735.543,E2 -19735.543} C_VEL
LIN {X 0,Y 248.514,Z 634.043,A -85,B 0,C 180,E1 -19736.903,E2 -19736.903} C_VEL
LIN {X 0,Y 250.257,Z 621.401,A -85,B 0,C 180,E1 -19738.06,E2 -19738.06} C_VEL
LIN {X 0,Y 251.759,Z 608.051,A -85,B 0,C 180,E1 -19738.901,E2 -19738.901} C_VEL
LIN {X 0,Y 252.653,Z 594.398,A -85,B 0,C 180,E1 -19739.416,E2 -19739.416} C_VEL
LIN {X 0,Y 254.921,Z 527.366,A -85,B 0,C 180,E1 -19741.279,E2 -19741.279} C_VEL
LIN {X 0,Y 251.063,Z 496.739,A -85,B 0,C 180,E1 -19742.831,E2 -19742.831} C_VEL
LIN {X 0,Y 249.796,Z 487.991,A -85,B 0,C 180,E1 -19743.338,E2 -19743.338} C_VEL
LIN {X 0,Y 251.744,Z 474.31,A -85,B 0,C 180,E1 -19745.893,E2 -19745.893} C_VEL
LIN {X 0,Y 251.661,Z 471.86,A -85,B 0,C 180,E1 -19746.425,E2 -19746.425} C_VEL
LIN {X 0,Y 249.054,Z 459.859,A -85,B 0,C 180,E1 -19749.543,E2 -19749.543} C_VEL
LIN {X 0,Y 245.988,Z 448.979,A -85,B 0,C 180,E1 -19752.635,E2 -19752.635} C_VEL
LIN {X 0,Y 242.568,Z 438.552,A -85,B 0,C 180,E1 -19755.944,E2 -19755.944} C_VEL
LIN {X 0,Y 238.975,Z 429.146,A -85,B 0,C 180,E1 -19759.129,E2 -19759.129} C_VEL
LIN {X 0,Y 235.94,Z 422.05,A -85,B 0,C 180,E1 -19761.823,E2 -19761.823} C_VEL
LIN {X 0,Y 234.954,Z 419.392,A -85,B 0,C 180,E1 -19762.921,E2 -19762.921} C_VEL
LIN {X 0,Y 234.954,Z 419.205,A -85,B 0,C 180,E1 -19767.424,E2 -19767.424} C_VEL
LIN {X 0,Y 234.898,Z 419.207,A -85,B 0,C 180,E1 -19771.399,E2 -19771.399} C_VEL
LIN {X 0,Y 234.955,Z 419.202,A -85,B 0,C 180,E1 -19775.243,E2 -19775.243} C_VEL
LIN {X 0,Y 234.943,Z 419.221,A -85,B 0,C 180,E1 -19778.963,E2 -19778.963} C_VEL
LIN {X 0,Y 235.052,Z 419.182,A -85,B 0,C 180,E1 -19783.098,E2 -19783.098} C_VEL
LIN {X 0,Y 235.088,Z 419.172,A -85,B 0,C 180,E1 -19787.921,E2 -19787.921} C_VEL
LIN {X 0,Y 235.318,Z 419.17,A -85,B 0,C 180,E1 -19791.412,E2 -19791.412} C_VEL
LIN {X 0,Y 235.355,Z 419.157,A -85,B 0,C 180,E1 -19793.14,E2 -19793.14} C_VEL
LIN {X 0,Y 235.203,Z 419.154,A -85,B 0,C 180,E1 -19795.781,E2 -19795.781} C_VEL
LIN {X 0,Y 234.627,Z 419.241,A -85,B 0,C 180,E1 -19797.214,E2 -19797.214} C_VEL
LIN {X 0,Y 231.904,Z 419.595,A -85,B 0,C 180,E1 -19799.555,E2 -19799.555} C_VEL
LIN {X 0,Y 228.629,Z 419.973,A -85,B 0,C 180,E1 -19802.442,E2 -19802.442} C_VEL
LIN {X 0,Y 228.218,Z 420.025,A -85,B 0,C 180,E1 -19803.441,E2 -19803.441} C_VEL
LIN {X 0,Y 228.302,Z 420.04,A -85,B 0,C 180,E1 -19807.073,E2 -19807.073} C_VEL
LIN {X 0,Y 228.128,Z 420.038,A -85,B 0,C 180,E1 -19810.652,E2 -19810.652} C_VEL
LIN {X 0,Y 228.002,Z 420.052,A -85,B 0,C 180,E1 -19816.106,E2 -19816.106} C_VEL
LIN {X 0,Y 227.921,Z 420.073,A -85,B 0,C 180,E1 -19821.717,E2 -19821.717} C_VEL
LIN {X 0,Y 227.903,Z 420.096,A -85,B 0,C 180,E1 -19826.581,E2 -19826.581} C_VEL
LIN {X 0,Y 227.872,Z 420.081,A -85,B 0,C 180,E1 -19830.279,E2 -19830.279} C_VEL
LIN {X 0,Y 227.878,Z 420.08,A -85,B 0,C 180,E1 -19833.72,E2 -19833.72} C_VEL
LIN {X 0,Y 227.841,Z 420.078,A -85,B 0,C 180,E1 -19838.092,E2 -19838.092} C_VEL
LIN {X 0,Y 227.826,Z 420.228,A -85,B 0,C 180,E1 -19842.572,E2 -19842.572} C_VEL
LIN {X 0,Y 228.032,Z 421.143,A -85,B 0,C 180,E1 -19842.992,E2 -19842.992} C_VEL
LIN {X 0,Y 229.013,Z 423.186,A -85,B 0,C 180,E1 -19843.668,E2 -19843.668} C_VEL
LIN {X 0,Y 229.985,Z 424.339,A -85,B 0,C 180,E1 -19844.155,E2 -19844.155} C_VEL
LIN {X 0,Y 238.299,Z 439.451,A -85,B 0,C 180,E1 -19848.513,E2 -19848.513} C_VEL
LIN {X 0,Y 239.705,Z 442.713,A -85,B 0,C 180,E1 -19849.28,E2 -19849.28} C_VEL
LIN {X 0,Y 243.328,Z 457.788,A -85,B 0,C 180,E1 -19852.008,E2 -19852.008} C_VEL
LIN {X 0,Y 245.099,Z 465.378,A -85,B 0,C 180,E1 -19853.278,E2 -19853.278} C_VEL
LIN {X 0,Y 244.153,Z 488.831,A -85,B 0,C 180,E1 -19856.022,E2 -19856.022} C_VEL
LIN {X 0,Y 247.438,Z 522.283,A -85,B 0,C 180,E1 -19857.666,E2 -19857.666} C_VEL
LIN {X 0,Y 248.243,Z 535.85,A -85,B 0,C 180,E1 -19858.236,E2 -19858.236} C_VEL
LIN {X 0,Y 245.918,Z 598.611,A -85,B 0,C 180,E1 -19859.991,E2 -19859.991} C_VEL
LIN {X 0,Y 245.02,Z 612.155,A -85,B 0,C 180,E1 -19860.521,E2 -19860.521} C_VEL
LIN {X 0,Y 243.515,Z 624.892,A -85,B 0,C 180,E1 -19861.327,E2 -19861.327} C_VEL
LIN {X 0,Y 241.932,Z 635.743,A -85,B 0,C 180,E1 -19862.303,E2 -19862.303} C_VEL
LIN {X 0,Y 239.874,Z 647.431,A -85,B 0,C 180,E1 -19863.695,E2 -19863.695} C_VEL
LIN {X 0,Y 237.321,Z 659.051,A -85,B 0,C 180,E1 -19865.506,E2 -19865.506} C_VEL
LIN {X 0,Y 234.845,Z 669.366,A -85,B 0,C 180,E1 -19867.569,E2 -19867.569} C_VEL
LIN {X 0,Y 232.654,Z 678.315,A -85,B 0,C 180,E1 -19869.866,E2 -19869.866} C_VEL
LIN {X 0,Y 230.619,Z 685.815,A -85,B 0,C 180,E1 -19872.257,E2 -19872.257} C_VEL
LIN {X 0,Y 228.738,Z 692.347,A -85,B 0,C 180,E1 -19874.861,E2 -19874.861} C_VEL
LIN {X 0,Y 227.455,Z 697.534,A -85,B 0,C 180,E1 -19877.509,E2 -19877.509} C_VEL
LIN {X 0,Y 226.513,Z 701.539,A -85,B 0,C 180,E1 -19880.174,E2 -19880.174} C_VEL
LIN {X 0,Y 225.947,Z 704.488,A -85,B 0,C 180,E1 -19882.853,E2 -19882.853} C_VEL
LIN {X 0,Y 225.711,Z 706.208,A -85,B 0,C 180,E1 -19885.13,E2 -19885.13} C_VEL
LIN {X 0,Y 225.658,Z 707.509,A -85,B 0,C 180,E1 -19888.215,E2 -19888.215} C_VEL
LIN {X 0,Y 225.706,Z 707.723,A -85,B 0,C 180,E1 -19890,E2 -19890} C_VEL
LIN {X 0,Y 225.691,Z 707.498,A -85,B 0,C 180,E1 -19891.784,E2 -19891.784} C_VEL
LIN {X 0,Y 225.717,Z 706.173,A -85,B 0,C 180,E1 -19894.887,E2 -19894.887} C_VEL
LIN {X 0,Y 225.95,Z 704.449,A -85,B 0,C 180,E1 -19897.147,E2 -19897.147} C_VEL
LIN {X 0,Y 226.515,Z 701.485,A -85,B 0,C 180,E1 -19899.825,E2 -19899.825} C_VEL
LIN {X 0,Y 227.457,Z 697.46,A -85,B 0,C 180,E1 -19902.491,E2 -19902.491} C_VEL
LIN {X 0,Y 229.034,Z 691.255,A -85,B 0,C 180,E1 -19905.575,E2 -19905.575} C_VEL
LIN {X 0,Y 230.989,Z 684.486,A -85,B 0,C 180,E1 -19908.171,E2 -19908.171} C_VEL
LIN {X 0,Y 233.123,Z 676.352,A -85,B 0,C 180,E1 -19910.645,E2 -19910.645} C_VEL
LIN {X 0,Y 235.298,Z 667.257,A -85,B 0,C 180,E1 -19912.848,E2 -19912.848} C_VEL
LIN {X 0,Y 237.883,Z 656.499,A -85,B 0,C 180,E1 -19914.898,E2 -19914.898} C_VEL
LIN {X 0,Y 240.148,Z 645.61,A -85,B 0,C 180,E1 -19916.506,E2 -19916.506} C_VEL
LIN {X 0,Y 241.36,Z 639.639,A -85,B 0,C 180,E1 -19917.298,E2 -19917.298} C_VEL
LIN {X 0,Y 246.205,Z 631.92,A -85,B 0,C 180,E1 -19919.499,E2 -19919.499} C_VEL
LIN {X 0,Y 251.754,Z 622.776,A -85,B 0,C 180,E1 -19921.562,E2 -19921.562} C_VEL
LIN {X 0,Y 257.888,Z 611.815,A -85,B 0,C 180,E1 -19923.494,E2 -19923.494} C_VEL
LIN {X 0,Y 264.035,Z 599.788,A -85,B 0,C 180,E1 -19925.142,E2 -19925.142} C_VEL
LIN {X 0,Y 269.935,Z 586.549,A -85,B 0,C 180,E1 -19926.553,E2 -19926.553} C_VEL
LIN {X 0,Y 275.592,Z 571.875,A -85,B 0,C 180,E1 -19927.737,E2 -19927.737} C_VEL
LIN {X 0,Y 280.32,Z 556.868,A -85,B 0,C 180,E1 -19928.669,E2 -19928.669} C_VEL
LIN {X 0,Y 284.071,Z 540.979,A -85,B 0,C 180,E1 -19929.487,E2 -19929.487} C_VEL
LIN {X 0,Y 285.701,Z 530.654,A -85,B 0,C 180,E1 -19930.259,E2 -19930.259} C_VEL
LIN {X 0,Y 287.427,Z 518.631,A -85,B 0,C 180,E1 -19931.452,E2 -19931.452} C_VEL
LIN {X 0,Y 288.795,Z 509.187,A -85,B 0,C 180,E1 -19932.602,E2 -19932.602} C_VEL
LIN {X 0,Y 288.741,Z 507.038,A -85,B 0,C 180,E1 -19933.394,E2 -19933.394} C_VEL
LIN {X 0,Y 288.787,Z 503.188,A -85,B 0,C 180,E1 -19935.44,E2 -19935.44} C_VEL
LIN {X 0,Y 289.169,Z 501.212,A -85,B 0,C 180,E1 -19937.116,E2 -19937.116} C_VEL
LIN {X 0,Y 290.132,Z 500.016,A -85,B 0,C 180,E1 -19939.153,E2 -19939.153} C_VEL
LIN {X 0,Y 291.653,Z 500.261,A -85,B 0,C 180,E1 -19941.206,E2 -19941.206} C_VEL
LIN {X 0,Y 286.861,Z 523.887,A -85,B 0,C 180,E1 -19942.521,E2 -19942.521} C_VEL
LIN {X 0,Y 283.771,Z 537.513,A -85,B 0,C 180,E1 -19943.53,E2 -19943.53} C_VEL
LIN {X 0,Y 279.902,Z 550.284,A -85,B 0,C 180,E1 -19944.725,E2 -19944.725} C_VEL
LIN {X 0,Y 275.748,Z 561.626,A -85,B 0,C 180,E1 -19946.115,E2 -19946.115} C_VEL
LIN {X 0,Y 271.618,Z 571.144,A -85,B 0,C 180,E1 -19947.527,E2 -19947.527} C_VEL
LIN {X 0,Y 267.144,Z 579.946,A -85,B 0,C 180,E1 -19949.136,E2 -19949.136} C_VEL
LIN {X 0,Y 262.054,Z 588.641,A -85,B 0,C 180,E1 -19951.135,E2 -19951.135} C_VEL
LIN {X 0,Y 257.282,Z 595.702,A -85,B 0,C 180,E1 -19953.21,E2 -19953.21} C_VEL
LIN {X 0,Y 252.816,Z 601.446,A -85,B 0,C 180,E1 -19955.356,E2 -19955.356} C_VEL
LIN {X 0,Y 248.637,Z 606.007,A -85,B 0,C 180,E1 -19957.568,E2 -19957.568} C_VEL
LIN {X 0,Y 244.784,Z 609.474,A -85,B 0,C 180,E1 -19959.847,E2 -19959.847} C_VEL
LIN {X 0,Y 242.453,Z 611.226,A -85,B 0,C 180,E1 -19961.406,E2 -19961.406} C_VEL
LIN {X 0,Y 240.242,Z 612.565,A -85,B 0,C 180,E1 -19962.99,E2 -19962.99} C_VEL
LIN {X 0,Y 238.298,Z 613.465,A -85,B 0,C 180,E1 -19964.607,E2 -19964.607} C_VEL
LIN {X 0,Y 236.44,Z 613.961,A -85,B 0,C 180,E1 -19966.244,E2 -19966.244} C_VEL
LIN {X 0,Y 234.754,Z 614.054,A -85,B 0,C 180,E1 -19967.903,E2 -19967.903} C_VEL
LIN {X 0,Y 231.97,Z 613.028,A -85,B 0,C 180,E1 -19971.287,E2 -19971.287} C_VEL
LIN {X 0,Y 231.018,Z 611.855,A -85,B 0,C 180,E1 -19973.011,E2 -19973.011} C_VEL
LIN {X 0,Y 230.216,Z 610.276,A -85,B 0,C 180,E1 -19974.745,E2 -19974.745} C_VEL
LIN {X 0,Y 229.031,Z 607.147,A -85,B 0,C 180,E1 -19977.362,E2 -19977.362} C_VEL
LIN {X 0,Y 228.13,Z 602.99,A -85,B 0,C 180,E1 -19980,E2 -19980} C_VEL
LIN {X 0,Y 227.838,Z 596.754,A -85,B 0,C 180,E1 -19983.095,E2 -19983.095} C_VEL
LIN {X 0,Y 227.841,Z 589.966,A -85,B 0,C 180,E1 -19985.754,E2 -19985.754} C_VEL
LIN {X 0,Y 228.287,Z 581.672,A -85,B 0,C 180,E1 -19988.409,E2 -19988.409} C_VEL
LIN {X 0,Y 228.84,Z 571.521,A -85,B 0,C 180,E1 -19991.067,E2 -19991.067} C_VEL
LIN {X 0,Y 229.534,Z 560.032,A -85,B 0,C 180,E1 -19993.501,E2 -19993.501} C_VEL
LIN {X 0,Y 230.208,Z 548.447,A -85,B 0,C 180,E1 -19995.494,E2 -19995.494} C_VEL
LIN {X 0,Y 231.018,Z 535.677,A -85,B 0,C 180,E1 -19997.254,E2 -19997.254} C_VEL
LIN {X 0,Y 231.797,Z 522.398,A -85,B 0,C 180,E1 -19998.678,E2 -19998.678} C_VEL
LIN {X 0,Y 232.241,Z 508.105,A -85,B 0,C 180,E1 -19999.836,E2 -19999.836} C_VEL
LIN {X 0,Y 232.839,Z 486.046,A -85,B 0,C 180,E1 -20001.03,E2 -20001.03} C_VEL
LIN {X 0,Y 234.117,Z 446.749,A -85,B 0,C 180,E1 -20003.004,E2 -20003.004} C_VEL
LIN {X 0,Y 234.052,Z 442.346,A -85,B 0,C 180,E1 -20003.234,E2 -20003.234} C_VEL
LIN {X 0,Y 228.142,Z 420.957,A -85,B 0,C 180,E1 -20004.613,E2 -20004.613} C_VEL
LIN {X 0,Y 227.984,Z 420.174,A -85,B 0,C 180,E1 -20004.922,E2 -20004.922} C_VEL
LIN {X 0,Y 227.875,Z 420.084,A -85,B 0,C 180,E1 -20010.281,E2 -20010.281} C_VEL
LIN {X 0,Y 227.91,Z 420.203,A -85,B 0,C 180,E1 -20015.323,E2 -20015.323} C_VEL
LIN {X 0,Y 228.086,Z 421.119,A -85,B 0,C 180,E1 -20015.835,E2 -20015.835} C_VEL
LIN {X 0,Y 231.525,Z 428.893,A -85,B 0,C 180,E1 -20019.041,E2 -20019.041} C_VEL
LIN {X 0,Y 235.024,Z 437.619,A -85,B 0,C 180,E1 -20022.286,E2 -20022.286} C_VEL
LIN {X 0,Y 239.002,Z 449.02,A -85,B 0,C 180,E1 -20026.091,E2 -20026.091} C_VEL
LIN {X 0,Y 242.124,Z 460.045,A -85,B 0,C 180,E1 -20029.383,E2 -20029.383} C_VEL
LIN {X 0,Y 245.114,Z 473.421,A -85,B 0,C 180,E1 -20032.978,E2 -20032.978} C_VEL
LIN {X 0,Y 245.456,Z 475.645,A -85,B 0,C 180,E1 -20033.534,E2 -20033.534} C_VEL
LIN {X 0,Y 243.667,Z 488.357,A -85,B 0,C 180,E1 -20035.885,E2 -20035.885} C_VEL
LIN {X 0,Y 247.362,Z 515.93,A -85,B 0,C 180,E1 -20037.407,E2 -20037.407} C_VEL
LIN {X 0,Y 248.862,Z 529.169,A -85,B 0,C 180,E1 -20038.071,E2 -20038.071} C_VEL
LIN {X 0,Y 246.034,Z 601.175,A -85,B 0,C 180,E1 -20040.125,E2 -20040.125} C_VEL
LIN {X 0,Y 244.769,Z 614.446,A -85,B 0,C 180,E1 -20040.783,E2 -20040.783} C_VEL
LIN {X 0,Y 243.046,Z 628.057,A -85,B 0,C 180,E1 -20041.855,E2 -20041.855} C_VEL
LIN {X 0,Y 241.08,Z 639.868,A -85,B 0,C 180,E1 -20043.137,E2 -20043.137} C_VEL
LIN {X 0,Y 238.804,Z 651.106,A -85,B 0,C 180,E1 -20044.74,E2 -20044.74} C_VEL
LIN {X 0,Y 236.452,Z 661.258,A -85,B 0,C 180,E1 -20046.575,E2 -20046.575} C_VEL
LIN {X 0,Y 234.359,Z 670.034,A -85,B 0,C 180,E1 -20048.568,E2 -20048.568} C_VEL
LIN {X 0,Y 232.087,Z 678.609,A -85,B 0,C 180,E1 -20051.003,E2 -20051.003} C_VEL
LIN {X 0,Y 229.965,Z 685.849,A -85,B 0,C 180,E1 -20053.579,E2 -20053.579} C_VEL
LIN {X 0,Y 228.164,Z 692.487,A -85,B 0,C 180,E1 -20056.643,E2 -20056.643} C_VEL
LIN {X 0,Y 227.028,Z 696.846,A -85,B 0,C 180,E1 -20059.296,E2 -20059.296} C_VEL
LIN {X 0,Y 226.492,Z 699.14,A -85,B 0,C 180,E1 -20061.075,E2 -20061.075} C_VEL
LIN {X 0,Y 226.083,Z 701.01,A -85,B 0,C 180,E1 -20062.857,E2 -20062.857} C_VEL
LIN {X 0,Y 225.711,Z 702.741,A -85,B 0,C 180,E1 -20065.135,E2 -20065.135} C_VEL
LIN {X 0,Y 225.597,Z 704.05,A -85,B 0,C 180,E1 -20068.215,E2 -20068.215} C_VEL
LIN {X 0,Y 225.638,Z 704.283,A -85,B 0,C 180,E1 -20070,E2 -20070} C_VEL
LIN {X 0,Y 225.596,Z 704.085,A -85,B 0,C 180,E1 -20071.785,E2 -20071.785} C_VEL
LIN {X 0,Y 225.741,Z 702.765,A -85,B 0,C 180,E1 -20074.956,E2 -20074.956} C_VEL
LIN {X 0,Y 226.026,Z 701.136,A -85,B 0,C 180,E1 -20077.145,E2 -20077.145} C_VEL
LIN {X 0,Y 226.7,Z 698.238,A -85,B 0,C 180,E1 -20079.818,E2 -20079.818} C_VEL
LIN {X 0,Y 227.667,Z 694.301,A -85,B 0,C 180,E1 -20082.48,E2 -20082.48} C_VEL
LIN {X 0,Y 229.04,Z 689.2,A -85,B 0,C 180,E1 -20085.119,E2 -20085.119} C_VEL
LIN {X 0,Y 230.915,Z 682.77,A -85,B 0,C 180,E1 -20087.72,E2 -20087.72} C_VEL
LIN {X 0,Y 233.141,Z 674.781,A -85,B 0,C 180,E1 -20090.284,E2 -20090.284} C_VEL
LIN {X 0,Y 235.248,Z 666.463,A -85,B 0,C 180,E1 -20092.429,E2 -20092.429} C_VEL
LIN {X 0,Y 237.602,Z 656.546,A -85,B 0,C 180,E1 -20094.463,E2 -20094.463} C_VEL
LIN {X 0,Y 240.14,Z 645.226,A -85,B 0,C 180,E1 -20096.274,E2 -20096.274} C_VEL
LIN {X 0,Y 242.191,Z 634.071,A -85,B 0,C 180,E1 -20097.665,E2 -20097.665} C_VEL
LIN {X 0,Y 244.031,Z 621.416,A -85,B 0,C 180,E1 -20098.842,E2 -20098.842} C_VEL
LIN {X 0,Y 245.515,Z 608.929,A -85,B 0,C 180,E1 -20099.649,E2 -20099.649} C_VEL
LIN {X 0,Y 246.42,Z 595.983,A -85,B 0,C 180,E1 -20100.177,E2 -20100.177} C_VEL
LIN {X 0,Y 248.867,Z 528.423,A -85,B 0,C 180,E1 -20102.091,E2 -20102.091} C_VEL
LIN {X 0,Y 245.24,Z 498.825,A -85,B 0,C 180,E1 -20103.638,E2 -20103.638} C_VEL
LIN {X 0,Y 243.707,Z 487.816,A -85,B 0,C 180,E1 -20104.305,E2 -20104.305} C_VEL
LIN {X 0,Y 245.511,Z 475.211,A -85,B 0,C 180,E1 -20106.723,E2 -20106.723} C_VEL
LIN {X 0,Y 243.013,Z 463.302,A -85,B 0,C 180,E1 -20109.856,E2 -20109.856} C_VEL
LIN {X 0,Y 240.113,Z 452.658,A -85,B 0,C 180,E1 -20112.967,E2 -20112.967} C_VEL
LIN {X 0,Y 236.763,Z 442.444,A -85,B 0,C 180,E1 -20116.242,E2 -20116.242} C_VEL
LIN {X 0,Y 233.542,Z 433.679,A -85,B 0,C 180,E1 -20119.326,E2 -20119.326} C_VEL
LIN {X 0,Y 229.569,Z 424.19,A -85,B 0,C 180,E1 -20123.013,E2 -20123.013} C_VEL
LIN {X 0,Y 227.911,Z 420.369,A -85,B 0,C 180,E1 -20124.677,E2 -20124.677} C_VEL
LIN {X 0,Y 227.895,Z 420.09,A -85,B 0,C 180,E1 -20125.213,E2 -20125.213} C_VEL
LIN {X 0,Y 227.875,Z 420.084,A -85,B 0,C 180,E1 -20130.431,E2 -20130.431} C_VEL
LIN {X 0,Y 227.904,Z 420.091,A -85,B 0,C 180,E1 -20134.423,E2 -20134.423} C_VEL
LIN {X 0,Y 227.927,Z 420.085,A -85,B 0,C 180,E1 -20138.283,E2 -20138.283} C_VEL
LIN {X 0,Y 228.012,Z 420.067,A -85,B 0,C 180,E1 -20143.894,E2 -20143.894} C_VEL
LIN {X 0,Y 228.128,Z 420.038,A -85,B 0,C 180,E1 -20149.348,E2 -20149.348} C_VEL
LIN {X 0,Y 228.307,Z 420.038,A -85,B 0,C 180,E1 -20152.927,E2 -20152.927} C_VEL
LIN {X 0,Y 228.536,Z 420.013,A -85,B 0,C 180,E1 -20158.238,E2 -20158.238} C_VEL
LIN {X 0,Y 228.535,Z 419.984,A -85,B 0,C 180,E1 -20161.762,E2 -20161.762} C_VEL
LIN {X 0,Y 228.218,Z 420.025,A -85,B 0,C 180,E1 -20163.441,E2 -20163.441} C_VEL
LIN {X 0,Y 227.438,Z 420.146,A -85,B 0,C 180,E1 -20164.913,E2 -20164.913} C_VEL
LIN {X 0,Y 224.589,Z 420.498,A -85,B 0,C 180,E1 -20167.319,E2 -20167.319} C_VEL
LIN {X 0,Y 221.388,Z 420.879,A -85,B 0,C 180,E1 -20170.289,E2 -20170.289} C_VEL
LIN {X 0,Y 221.023,Z 420.928,A -85,B 0,C 180,E1 -20171.317,E2 -20171.317} C_VEL
LIN {X 0,Y 220.968,Z 420.927,A -85,B 0,C 180,E1 -20176.634,E2 -20176.634} C_VEL
LIN {X 0,Y 220.847,Z 420.973,A -85,B 0,C 180,E1 -20180.491,E2 -20180.491} C_VEL
LIN {X 0,Y 220.798,Z 420.959,A -85,B 0,C 180,E1 -20184.443,E2 -20184.443} C_VEL
LIN {X 0,Y 220.797,Z 420.957,A -85,B 0,C 180,E1 -20188.519,E2 -20188.519} C_VEL
LIN {X 0,Y 220.813,Z 420.969,A -85,B 0,C 180,E1 -20192.757,E2 -20192.757} C_VEL
LIN {X 0,Y 220.804,Z 420.977,A -85,B 0,C 180,E1 -20197.275,E2 -20197.275} C_VEL
LIN {X 0,Y 220.796,Z 421.09,A -85,B 0,C 180,E1 -20200.377,E2 -20200.377} C_VEL
LIN {X 0,Y 221.009,Z 422.179,A -85,B 0,C 180,E1 -20200.928,E2 -20200.928} C_VEL
LIN {X 0,Y 222.009,Z 424.229,A -85,B 0,C 180,E1 -20201.666,E2 -20201.666} C_VEL
LIN {X 0,Y 223.127,Z 425.43,A -85,B 0,C 180,E1 -20202.254,E2 -20202.254} C_VEL
LIN {X 0,Y 228.487,Z 435.29,A -85,B 0,C 180,E1 -20205.48,E2 -20205.48} C_VEL
LIN {X 0,Y 233.586,Z 444.551,A -85,B 0,C 180,E1 -20208.13,E2 -20208.13} C_VEL
LIN {X 0,Y 234.638,Z 447.423,A -85,B 0,C 180,E1 -20208.779,E2 -20208.779} C_VEL
LIN {X 0,Y 238.949,Z 466.18,A -85,B 0,C 180,E1 -20212.228,E2 -20212.228} C_VEL
LIN {X 0,Y 239.244,Z 467.663,A -85,B 0,C 180,E1 -20212.481,E2 -20212.481} C_VEL
LIN {X 0,Y 238.183,Z 488.902,A -85,B 0,C 180,E1 -20215.048,E2 -20215.048} C_VEL
LIN {X 0,Y 241.422,Z 522.783,A -85,B 0,C 180,E1 -20216.772,E2 -20216.772} C_VEL
LIN {X 0,Y 242.242,Z 535.747,A -85,B 0,C 180,E1 -20217.346,E2 -20217.346} C_VEL
LIN {X 0,Y 239.687,Z 600.371,A -85,B 0,C 180,E1 -20219.188,E2 -20219.188} C_VEL
LIN {X 0,Y 238.688,Z 613.924,A -85,B 0,C 180,E1 -20219.78,E2 -20219.78} C_VEL
LIN {X 0,Y 237.142,Z 626.143,A -85,B 0,C 180,E1 -20220.603,E2 -20220.603} C_VEL
LIN {X 0,Y 235.383,Z 637.617,A -85,B 0,C 180,E1 -20221.706,E2 -20221.706} C_VEL
LIN {X 0,Y 233.226,Z 648.801,A -85,B 0,C 180,E1 -20223.127,E2 -20223.127} C_VEL
LIN {X 0,Y 230.593,Z 660.169,A -85,B 0,C 180,E1 -20224.983,E2 -20224.983} C_VEL
LIN {X 0,Y 228.275,Z 669.321,A -85,B 0,C 180,E1 -20226.887,E2 -20226.887} C_VEL
LIN {X 0,Y 225.838,Z 678.809,A -85,B 0,C 180,E1 -20229.406,E2 -20229.406} C_VEL
LIN {X 0,Y 223.503,Z 686.983,A -85,B 0,C 180,E1 -20232.146,E2 -20232.146} C_VEL
LIN {X 0,Y 221.866,Z 692.296,A -85,B 0,C 180,E1 -20234.38,E2 -20234.38} C_VEL
LIN {X 0,Y 220.509,Z 697.483,A -85,B 0,C 180,E1 -20237.108,E2 -20237.108} C_VEL
LIN {X 0,Y 219.513,Z 701.486,A -85,B 0,C 180,E1 -20239.858,E2 -20239.858} C_VEL
LIN {X 0,Y 218.876,Z 704.435,A -85,B 0,C 180,E1 -20242.62,E2 -20242.62} C_VEL
LIN {X 0,Y 218.596,Z 706.368,A -85,B 0,C 180,E1 -20245.324,E2 -20245.324} C_VEL
LIN {X 0,Y 218.558,Z 707.455,A -85,B 0,C 180,E1 -20248.157,E2 -20248.157} C_VEL
LIN {X 0,Y 218.622,Z 707.669,A -85,B 0,C 180,E1 -20250,E2 -20250} C_VEL
LIN {X 0,Y 218.589,Z 707.444,A -85,B 0,C 180,E1 -20251.842,E2 -20251.842} C_VEL
LIN {X 0,Y 218.622,Z 706.293,A -85,B 0,C 180,E1 -20254.757,E2 -20254.757} C_VEL
LIN {X 0,Y 218.879,Z 704.394,A -85,B 0,C 180,E1 -20257.379,E2 -20257.379} C_VEL
LIN {X 0,Y 219.515,Z 701.43,A -85,B 0,C 180,E1 -20260.142,E2 -20260.142} C_VEL
LIN {X 0,Y 220.511,Z 697.406,A -85,B 0,C 180,E1 -20262.891,E2 -20262.891} C_VEL
LIN {X 0,Y 222.196,Z 691.202,A -85,B 0,C 180,E1 -20266.067,E2 -20266.067} C_VEL
LIN {X 0,Y 224.214,Z 684.433,A -85,B 0,C 180,E1 -20268.741,E2 -20268.741} C_VEL
LIN {X 0,Y 226.333,Z 676.87,A -85,B 0,C 180,E1 -20271.123,E2 -20271.123} C_VEL
LIN {X 0,Y 228.746,Z 667.207,A -85,B 0,C 180,E1 -20273.541,E2 -20273.541} C_VEL
LIN {X 0,Y 231.45,Z 656.452,A -85,B 0,C 180,E1 -20275.639,E2 -20275.639} C_VEL
LIN {X 0,Y 233.823,Z 645.58,A -85,B 0,C 180,E1 -20277.282,E2 -20277.282} C_VEL
LIN {X 0,Y 234.75,Z 641.025,A -85,B 0,C 180,E1 -20277.891,E2 -20277.891} C_VEL
LIN {X 0,Y 240.133,Z 633.255,A -85,B 0,C 180,E1 -20280.322,E2 -20280.322} C_VEL
LIN {X 0,Y 245.825,Z 624.715,A -85,B 0,C 180,E1 -20282.415,E2 -20282.415} C_VEL
LIN {X 0,Y 252.139,Z 614.547,A -85,B 0,C 180,E1 -20284.363,E2 -20284.363} C_VEL
LIN {X 0,Y 258.425,Z 603.482,A -85,B 0,C 180,E1 -20286.022,E2 -20286.022} C_VEL
LIN {X 0,Y 264.433,Z 591.525,A -85,B 0,C 180,E1 -20287.442,E2 -20287.442} C_VEL
LIN {X 0,Y 270.265,Z 578.503,A -85,B 0,C 180,E1 -20288.616,E2 -20288.616} C_VEL
LIN {X 0,Y 275.528,Z 564.454,A -85,B 0,C 180,E1 -20289.619,E2 -20289.619} C_VEL
LIN {X 0,Y 280.447,Z 548.136,A -85,B 0,C 180,E1 -20290.506,E2 -20290.506} C_VEL
LIN {X 0,Y 282.142,Z 540.68,A -85,B 0,C 180,E1 -20290.934,E2 -20290.934} C_VEL
LIN {X 0,Y 284.117,Z 529.544,A -85,B 0,C 180,E1 -20291.844,E2 -20291.844} C_VEL
LIN {X 0,Y 286.166,Z 517.414,A -85,B 0,C 180,E1 -20293.157,E2 -20293.157} C_VEL
LIN {X 0,Y 286.769,Z 513.897,A -85,B 0,C 180,E1 -20293.646,E2 -20293.646} C_VEL
LIN {X 0,Y 286.981,Z 509.727,A -85,B 0,C 180,E1 -20295.856,E2 -20295.856} C_VEL
LIN {X 0,Y 287.472,Z 507.89,A -85,B 0,C 180,E1 -20297.481,E2 -20297.481} C_VEL
LIN {X 0,Y 288.282,Z 506.92,A -85,B 0,C 180,E1 -20299.091,E2 -20299.091} C_VEL
LIN {X 0,Y 288.952,Z 506.899,A -85,B 0,C 180,E1 -20300.139,E2 -20300.139} C_VEL
LIN {X 0,Y 284.735,Z 526.4,A -85,B 0,C 180,E1 -20301.256,E2 -20301.256} C_VEL
LIN {X 0,Y 281.372,Z 539.943,A -85,B 0,C 180,E1 -20302.269,E2 -20302.269} C_VEL
LIN {X 0,Y 277.281,Z 552.399,A -85,B 0,C 180,E1 -20303.442,E2 -20303.442} C_VEL
LIN {X 0,Y 272.383,Z 564.598,A -85,B 0,C 180,E1 -20304.964,E2 -20304.964} C_VEL
LIN {X 0,Y 267.516,Z 574.699,A -85,B 0,C 180,E1 -20306.516,E2 -20306.516} C_VEL
LIN {X 0,Y 261.88,Z 584.645,A -85,B 0,C 180,E1 -20308.445,E2 -20308.445} C_VEL
LIN {X 0,Y 256.602,Z 592.628,A -85,B 0,C 180,E1 -20310.462,E2 -20310.462} C_VEL
LIN {X 0,Y 251.614,Z 599.178,A -85,B 0,C 180,E1 -20312.557,E2 -20312.557} C_VEL
LIN {X 0,Y 246.905,Z 604.458,A -85,B 0,C 180,E1 -20314.725,E2 -20314.725} C_VEL
LIN {X 0,Y 242.496,Z 608.646,A -85,B 0,C 180,E1 -20316.967,E2 -20316.967} C_VEL
LIN {X 0,Y 238.487,Z 611.785,A -85,B 0,C 180,E1 -20319.291,E2 -20319.291} C_VEL
LIN {X 0,Y 236.028,Z 613.327,A -85,B 0,C 180,E1 -20320.881,E2 -20320.881} C_VEL
LIN {X 0,Y 233.704,Z 614.46,A -85,B 0,C 180,E1 -20322.499,E2 -20322.499} C_VEL
LIN {X 0,Y 229.711,Z 615.469,A -85,B 0,C 180,E1 -20325.832,E2 -20325.832} C_VEL
LIN {X 0,Y 227.955,Z 615.389,A -85,B 0,C 180,E1 -20327.537,E2 -20327.537} C_VEL
LIN {X 0,Y 226.418,Z 614.878,A -85,B 0,C 180,E1 -20329.267,E2 -20329.267} C_VEL
LIN {X 0,Y 225.029,Z 613.959,A -85,B 0,C 180,E1 -20331.016,E2 -20331.016} C_VEL
LIN {X 0,Y 223.183,Z 610.894,A -85,B 0,C 180,E1 -20334.579,E2 -20334.579} C_VEL
LIN {X 0,Y 221.968,Z 607.505,A -85,B 0,C 180,E1 -20337.278,E2 -20337.278} C_VEL
LIN {X 0,Y 221.033,Z 603.052,A -85,B 0,C 180,E1 -20340,E2 -20340} C_VEL
LIN {X 0,Y 220.727,Z 596.389,A -85,B 0,C 180,E1 -20343.194,E2 -20343.194} C_VEL
LIN {X 0,Y 220.748,Z 589.299,A -85,B 0,C 180,E1 -20345.939,E2 -20345.939} C_VEL
LIN {X 0,Y 221.227,Z 580.663,A -85,B 0,C 180,E1 -20348.679,E2 -20348.679} C_VEL
LIN {X 0,Y 221.835,Z 569.95,A -85,B 0,C 180,E1 -20351.421,E2 -20351.421} C_VEL
LIN {X 0,Y 222.483,Z 559.002,A -85,B 0,C 180,E1 -20353.705,E2 -20353.705} C_VEL
LIN {X 0,Y 223.202,Z 546.939,A -85,B 0,C 180,E1 -20355.758,E2 -20355.758} C_VEL
LIN {X 0,Y 224.078,Z 533.561,A -85,B 0,C 180,E1 -20357.571,E2 -20357.571} C_VEL
LIN {X 0,Y 224.825,Z 519.528,A -85,B 0,C 180,E1 -20359.043,E2 -20359.043} C_VEL
LIN {X 0,Y 225.265,Z 504.901,A -85,B 0,C 180,E1 -20360.168,E2 -20360.168} C_VEL
LIN {X 0,Y 227.142,Z 445.905,A -85,B 0,C 180,E1 -20363.277,E2 -20363.277} C_VEL
LIN {X 0,Y 226.956,Z 443.34,A -85,B 0,C 180,E1 -20363.42,E2 -20363.42} C_VEL
LIN {X 0,Y 221.055,Z 421.704,A -85,B 0,C 180,E1 -20364.868,E2 -20364.868} C_VEL
LIN {X 0,Y 220.953,Z 421.038,A -85,B 0,C 180,E1 -20365.177,E2 -20365.177} C_VEL
LIN {X 0,Y 220.819,Z 420.969,A -85,B 0,C 180,E1 -20370.759,E2 -20370.759} C_VEL
LIN {X 0,Y 220.874,Z 421.188,A -85,B 0,C 180,E1 -20373.448,E2 -20373.448} C_VEL
LIN {X 0,Y 221.952,Z 423.927,A -85,B 0,C 180,E1 -20374.748,E2 -20374.748} C_VEL
LIN {X 0,Y 225.841,Z 432.629,A -85,B 0,C 180,E1 -20378.491,E2 -20378.491} C_VEL
LIN {X 0,Y 229.741,Z 442.634,A -85,B 0,C 180,E1 -20382.299,E2 -20382.299} C_VEL
LIN {X 0,Y 233.121,Z 452.637,A -85,B 0,C 180,E1 -20385.692,E2 -20385.692} C_VEL
LIN {X 0,Y 236.198,Z 463.832,A -85,B 0,C 180,E1 -20389.11,E2 -20389.11} C_VEL
LIN {X 0,Y 238.653,Z 474.829,A -85,B 0,C 180,E1 -20392.149,E2 -20392.149} C_VEL
LIN {X 0,Y 239.129,Z 477.611,A -85,B 0,C 180,E1 -20392.903,E2 -20392.903} C_VEL
LIN {X 0,Y 237.614,Z 488.419,A -85,B 0,C 180,E1 -20394.895,E2 -20394.895} C_VEL
LIN {X 0,Y 240.813,Z 512.38,A -85,B 0,C 180,E1 -20396.282,E2 -20396.282} C_VEL
LIN {X 0,Y 242.821,Z 530.167,A -85,B 0,C 180,E1 -20397.214,E2 -20397.214} C_VEL
LIN {X 0,Y 239.907,Z 601.168,A -85,B 0,C 180,E1 -20399.281,E2 -20399.281} C_VEL
LIN {X 0,Y 238.712,Z 613.743,A -85,B 0,C 180,E1 -20399.906,E2 -20399.906} C_VEL
LIN {X 0,Y 236.984,Z 627.015,A -85,B 0,C 180,E1 -20400.947,E2 -20400.947} C_VEL
LIN {X 0,Y 235.121,Z 638.271,A -85,B 0,C 180,E1 -20402.157,E2 -20402.157} C_VEL
LIN {X 0,Y 232.968,Z 648.617,A -85,B 0,C 180,E1 -20403.579,E2 -20403.579} C_VEL
LIN {X 0,Y 230.449,Z 659.223,A -85,B 0,C 180,E1 -20405.448,E2 -20405.448} C_VEL
LIN {X 0,Y 228.049,Z 668.829,A -85,B 0,C 180,E1 -20407.599,E2 -20407.599} C_VEL
LIN {X 0,Y 225.743,Z 677.32,A -85,B 0,C 180,E1 -20409.973,E2 -20409.973} C_VEL
LIN {X 0,Y 223.512,Z 684.806,A -85,B 0,C 180,E1 -20412.62,E2 -20412.62} C_VEL
LIN {X 0,Y 221.723,Z 690.812,A -85,B 0,C 180,E1 -20415.311,E2 -20415.311} C_VEL
LIN {X 0,Y 220.388,Z 695.562,A -85,B 0,C 180,E1 -20418.037,E2 -20418.037} C_VEL
LIN {X 0,Y 219.467,Z 699.194,A -85,B 0,C 180,E1 -20420.787,E2 -20420.787} C_VEL
LIN {X 0,Y 219.038,Z 701.065,A -85,B 0,C 180,E1 -20422.626,E2 -20422.626} C_VEL
LIN {X 0,Y 218.594,Z 703.009,A -85,B 0,C 180,E1 -20425.333,E2 -20425.333} C_VEL
LIN {X 0,Y 218.501,Z 704.105,A -85,B 0,C 180,E1 -20428.157,E2 -20428.157} C_VEL
LIN {X 0,Y 218.537,Z 704.337,A -85,B 0,C 180,E1 -20430,E2 -20430} C_VEL
LIN {X 0,Y 218.501,Z 704.139,A -85,B 0,C 180,E1 -20431.843,E2 -20431.843} C_VEL
LIN {X 0,Y 218.644,Z 702.993,A -85,B 0,C 180,E1 -20434.825,E2 -20434.825} C_VEL
LIN {X 0,Y 218.969,Z 701.189,A -85,B 0,C 180,E1 -20437.376,E2 -20437.376} C_VEL
LIN {X 0,Y 219.702,Z 698.29,A -85,B 0,C 180,E1 -20440.134,E2 -20440.134} C_VEL
LIN {X 0,Y 220.713,Z 694.353,A -85,B 0,C 180,E1 -20442.88,E2 -20442.88} C_VEL
LIN {X 0,Y 222.176,Z 689.25,A -85,B 0,C 180,E1 -20445.598,E2 -20445.598} C_VEL
LIN {X 0,Y 224.159,Z 682.819,A -85,B 0,C 180,E1 -20448.272,E2 -20448.272} C_VEL
LIN {X 0,Y 226.48,Z 674.828,A -85,B 0,C 180,E1 -20450.908,E2 -20450.908} C_VEL
LIN {X 0,Y 228.772,Z 666.159,A -85,B 0,C 180,E1 -20453.194,E2 -20453.194} C_VEL
LIN {X 0,Y 231.145,Z 656.587,A -85,B 0,C 180,E1 -20455.194,E2 -20455.194} C_VEL
LIN {X 0,Y 233.792,Z 645.262,A -85,B 0,C 180,E1 -20457.044,E2 -20457.044} C_VEL
LIN {X 0,Y 235.929,Z 634.099,A -85,B 0,C 180,E1 -20458.465,E2 -20458.465} C_VEL
LIN {X 0,Y 237.835,Z 621.432,A -85,B 0,C 180,E1 -20459.668,E2 -20459.668} C_VEL
LIN {X 0,Y 239.385,Z 608.925,A -85,B 0,C 180,E1 -20460.488,E2 -20460.488} C_VEL
LIN {X 0,Y 240.319,Z 595.916,A -85,B 0,C 180,E1 -20461.027,E2 -20461.027} C_VEL
LIN {X 0,Y 242.863,Z 529.513,A -85,B 0,C 180,E1 -20462.943,E2 -20462.943} C_VEL
LIN {X 0,Y 239.535,Z 501.37,A -85,B 0,C 180,E1 -20464.457,E2 -20464.457} C_VEL
LIN {X 0,Y 237.657,Z 487.987,A -85,B 0,C 180,E1 -20465.278,E2 -20465.278} C_VEL
LIN {X 0,Y 239.224,Z 477.823,A -85,B 0,C 180,E1 -20467.227,E2 -20467.227} C_VEL
LIN {X 0,Y 236.933,Z 466.561,A -85,B 0,C 180,E1 -20470.258,E2 -20470.258} C_VEL
LIN {X 0,Y 234.231,Z 456.359,A -85,B 0,C 180,E1 -20473.315,E2 -20473.315} C_VEL
LIN {X 0,Y 231.177,Z 446.857,A -85,B 0,C 180,E1 -20476.402,E2 -20476.402} C_VEL
LIN {X 0,Y 227.985,Z 437.893,A -85,B 0,C 180,E1 -20479.657,E2 -20479.657} C_VEL
LIN {X 0,Y 224.069,Z 428.435,A -85,B 0,C 180,E1 -20483.42,E2 -20483.42} C_VEL
LIN {X 0,Y 220.839,Z 421.171,A -85,B 0,C 180,E1 -20486.781,E2 -20486.781} C_VEL
LIN {X 0,Y 220.837,Z 420.972,A -85,B 0,C 180,E1 -20489.39,E2 -20489.39} C_VEL
LIN {X 0,Y 220.877,Z 420.974,A -85,B 0,C 180,E1 -20493.547,E2 -20493.547} C_VEL
LIN {X 0,Y 220.856,Z 420.956,A -85,B 0,C 180,E1 -20497.551,E2 -20497.551} C_VEL
LIN {X 0,Y 220.918,Z 420.939,A -85,B 0,C 180,E1 -20502.629,E2 -20502.629} C_VEL
LIN {X 0,Y 220.979,Z 420.935,A -85,B 0,C 180,E1 -20507.136,E2 -20507.136} C_VEL
LIN {X 0,Y 221.197,Z 420.92,A -85,B 0,C 180,E1 -20510.859,E2 -20510.859} C_VEL
LIN {X 0,Y 221.245,Z 420.92,A -85,B 0,C 180,E1 -20512.7,E2 -20512.7} C_VEL
LIN {X 0,Y 221.47,Z 420.892,A -85,B 0,C 180,E1 -20518.181,E2 -20518.181} C_VEL
LIN {X 0,Y 221.468,Z 420.864,A -85,B 0,C 180,E1 -20521.818,E2 -20521.818} C_VEL
LIN {X 0,Y 221.239,Z 420.915,A -85,B 0,C 180,E1 -20527.3,E2 -20527.3} C_VEL
LIN {X 0,Y 221.023,Z 420.928,A -85,B 0,C 180,E1 -20531.317,E2 -20531.317} C_VEL
LIN {X 0,Y 220.276,Z 421.046,A -85,B 0,C 180,E1 -20532.836,E2 -20532.836} C_VEL
LIN {X 0,Y 217.39,Z 421.412,A -85,B 0,C 180,E1 -20535.315,E2 -20535.315} C_VEL
LIN {X 0,Y 214.129,Z 421.812,A -85,B 0,C 180,E1 -20538.381,E2 -20538.381} C_VEL
LIN {X 0,Y 213.774,Z 421.847,A -85,B 0,C 180,E1 -20539.444,E2 -20539.444} C_VEL
LIN {X 0,Y 213.766,Z 421.827,A -85,B 0,C 180,E1 -20543.236,E2 -20543.236} C_VEL
LIN {X 0,Y 213.787,Z 421.839,A -85,B 0,C 180,E1 -20547.426,E2 -20547.426} C_VEL
LIN {X 0,Y 213.76,Z 421.859,A -85,B 0,C 180,E1 -20551.739,E2 -20551.739} C_VEL
LIN {X 0,Y 213.743,Z 421.852,A -85,B 0,C 180,E1 -20556.289,E2 -20556.289} C_VEL
LIN {X 0,Y 213.755,Z 422.041,A -85,B 0,C 180,E1 -20558.042,E2 -20558.042} C_VEL
LIN {X 0,Y 214.007,Z 423.135,A -85,B 0,C 180,E1 -20558.606,E2 -20558.606} C_VEL
LIN {X 0,Y 215.265,Z 425.353,A -85,B 0,C 180,E1 -20559.542,E2 -20559.542} C_VEL
LIN {X 0,Y 216.295,Z 426.632,A -85,B 0,C 180,E1 -20560.173,E2 -20560.173} C_VEL
LIN {X 0,Y 217.266,Z 428.921,A -85,B 0,C 180,E1 -20560.966,E2 -20560.966} C_VEL
LIN {X 0,Y 219.326,Z 432.237,A -85,B 0,C 180,E1 -20562.293,E2 -20562.293} C_VEL
LIN {X 0,Y 225.369,Z 442.966,A -85,B 0,C 180,E1 -20565.827,E2 -20565.827} C_VEL
LIN {X 0,Y 229.135,Z 450.35,A -85,B 0,C 180,E1 -20567.89,E2 -20567.89} C_VEL
LIN {X 0,Y 233.306,Z 469.448,A -85,B 0,C 180,E1 -20571.556,E2 -20571.556} C_VEL
LIN {X 0,Y 232.816,Z 479.556,A -85,B 0,C 180,E1 -20572.861,E2 -20572.861} C_VEL
LIN {X 0,Y 232.297,Z 488.888,A -85,B 0,C 180,E1 -20574.023,E2 -20574.023} C_VEL
LIN {X 0,Y 235.192,Z 520.15,A -85,B 0,C 180,E1 -20575.674,E2 -20575.674} C_VEL
LIN {X 0,Y 236.286,Z 536.303,A -85,B 0,C 180,E1 -20576.433,E2 -20576.433} C_VEL
LIN {X 0,Y 233.634,Z 600.424,A -85,B 0,C 180,E1 -20578.299,E2 -20578.299} C_VEL
LIN {X 0,Y 232.595,Z 613.928,A -85,B 0,C 180,E1 -20578.902,E2 -20578.902} C_VEL
LIN {X 0,Y 230.996,Z 626.126,A -85,B 0,C 180,E1 -20579.741,E2 -20579.741} C_VEL
LIN {X 0,Y 229.154,Z 637.587,A -85,B 0,C 180,E1 -20580.864,E2 -20580.864} C_VEL
LIN {X 0,Y 226.904,Z 648.765,A -85,B 0,C 180,E1 -20582.315,E2 -20582.315} C_VEL
LIN {X 0,Y 224.177,Z 660.128,A -85,B 0,C 180,E1 -20584.215,E2 -20584.215} C_VEL
LIN {X 0,Y 221.75,Z 669.276,A -85,B 0,C 180,E1 -20586.165,E2 -20586.165} C_VEL
LIN {X 0,Y 219.551,Z 677.526,A -85,B 0,C 180,E1 -20588.375,E2 -20588.375} C_VEL
LIN {X 0,Y 217.087,Z 685.716,A -85,B 0,C 180,E1 -20591.11,E2 -20591.11} C_VEL
LIN {X 0,Y 215.023,Z 692.245,A -85,B 0,C 180,E1 -20593.869,E2 -20593.869} C_VEL
LIN {X 0,Y 213.557,Z 697.431,A -85,B 0,C 180,E1 -20596.681,E2 -20596.681} C_VEL
LIN {X 0,Y 212.495,Z 701.433,A -85,B 0,C 180,E1 -20599.519,E2 -20599.519} C_VEL
LIN {X 0,Y 211.831,Z 704.381,A -85,B 0,C 180,E1 -20602.373,E2 -20602.373} C_VEL
LIN {X 0,Y 211.507,Z 706.475,A -85,B 0,C 180,E1 -20605.45,E2 -20605.45} C_VEL
LIN {X 0,Y 211.461,Z 707.401,A -85,B 0,C 180,E1 -20608.095,E2 -20608.095} C_VEL
LIN {X 0,Y 211.52,Z 707.615,A -85,B 0,C 180,E1 -20610,E2 -20610} C_VEL
LIN {X 0,Y 211.491,Z 707.39,A -85,B 0,C 180,E1 -20611.904,E2 -20611.904} C_VEL
LIN {X 0,Y 211.542,Z 706.384,A -85,B 0,C 180,E1 -20614.669,E2 -20614.669} C_VEL
LIN {X 0,Y 211.834,Z 704.34,A -85,B 0,C 180,E1 -20617.626,E2 -20617.626} C_VEL
LIN {X 0,Y 212.497,Z 701.376,A -85,B 0,C 180,E1 -20620.48,E2 -20620.48} C_VEL
LIN {X 0,Y 213.56,Z 697.352,A -85,B 0,C 180,E1 -20623.318,E2 -20623.318} C_VEL
LIN {X 0,Y 215.374,Z 691.148,A -85,B 0,C 180,E1 -20626.59,E2 -20626.59} C_VEL
LIN {X 0,Y 217.466,Z 684.38,A -85,B 0,C 180,E1 -20629.345,E2 -20629.345} C_VEL
LIN {X 0,Y 219.554,Z 677.368,A -85,B 0,C 180,E1 -20631.628,E2 -20631.628} C_VEL
LIN {X 0,Y 221.739,Z 669.081,A -85,B 0,C 180,E1 -20633.835,E2 -20633.835} C_VEL
LIN {X 0,Y 224.454,Z 658.727,A -85,B 0,C 180,E1 -20635.999,E2 -20635.999} C_VEL
LIN {X 0,Y 226.886,Z 648.477,A -85,B 0,C 180,E1 -20637.687,E2 -20637.687} C_VEL
LIN {X 0,Y 228.346,Z 641.973,A -85,B 0,C 180,E1 -20638.619,E2 -20638.619} C_VEL
LIN {X 0,Y 234.112,Z 634.494,A -85,B 0,C 180,E1 -20641.188,E2 -20641.188} C_VEL
LIN {X 0,Y 239.947,Z 626.551,A -85,B 0,C 180,E1 -20643.311,E2 -20643.311} C_VEL
LIN {X 0,Y 247.559,Z 615.431,A -85,B 0,C 180,E1 -20645.59,E2 -20645.59} C_VEL
LIN {X 0,Y 254.69,Z 603.865,A -85,B 0,C 180,E1 -20647.378,E2 -20647.378} C_VEL
LIN {X 0,Y 261.576,Z 591.221,A -85,B 0,C 180,E1 -20648.906,E2 -20648.906} C_VEL
LIN {X 0,Y 268.086,Z 577.553,A -85,B 0,C 180,E1 -20650.122,E2 -20650.122} C_VEL
LIN {X 0,Y 273.124,Z 565.12,A -85,B 0,C 180,E1 -20651.008,E2 -20651.008} C_VEL
LIN {X 0,Y 278.428,Z 549.144,A -85,B 0,C 180,E1 -20651.887,E2 -20651.887} C_VEL
LIN {X 0,Y 280.357,Z 541.672,A -85,B 0,C 180,E1 -20652.332,E2 -20652.332} C_VEL
LIN {X 0,Y 282.329,Z 531.957,A -85,B 0,C 180,E1 -20653.15,E2 -20653.15} C_VEL
LIN {X 0,Y 284.714,Z 519.972,A -85,B 0,C 180,E1 -20654.474,E2 -20654.474} C_VEL
LIN {X 0,Y 284.832,Z 519.262,A -85,B 0,C 180,E1 -20654.636,E2 -20654.636} C_VEL
LIN {X 0,Y 285.283,Z 515.937,A -85,B 0,C 180,E1 -20656.493,E2 -20656.493} C_VEL
LIN {X 0,Y 285.962,Z 514.282,A -85,B 0,C 180,E1 -20658.213,E2 -20658.213} C_VEL
LIN {X 0,Y 286.453,Z 513.794,A -85,B 0,C 180,E1 -20659.055,E2 -20659.055} C_VEL
LIN {X 0,Y 282.448,Z 531.125,A -85,B 0,C 180,E1 -20660.102,E2 -20660.102} C_VEL
LIN {X 0,Y 278.644,Z 544.378,A -85,B 0,C 180,E1 -20661.141,E2 -20661.141} C_VEL
LIN {X 0,Y 274.363,Z 556.106,A -85,B 0,C 180,E1 -20662.296,E2 -20662.296} C_VEL
LIN {X 0,Y 269.195,Z 567.77,A -85,B 0,C 180,E1 -20663.795,E2 -20663.795} C_VEL
LIN {X 0,Y 263.54,Z 578.337,A -85,B 0,C 180,E1 -20665.48,E2 -20665.48} C_VEL
LIN {X 0,Y 257.604,Z 587.792,A -85,B 0,C 180,E1 -20667.396,E2 -20667.396} C_VEL
LIN {X 0,Y 251.162,Z 596.602,A -85,B 0,C 180,E1 -20669.756,E2 -20669.756} C_VEL
LIN {X 0,Y 245.947,Z 602.593,A -85,B 0,C 180,E1 -20671.869,E2 -20671.869} C_VEL
LIN {X 0,Y 241.021,Z 607.469,A -85,B 0,C 180,E1 -20674.063,E2 -20674.063} C_VEL
LIN {X 0,Y 236.405,Z 611.256,A -85,B 0,C 180,E1 -20676.338,E2 -20676.338} C_VEL
LIN {X 0,Y 232.197,Z 614.044,A -85,B 0,C 180,E1 -20678.703,E2 -20678.703} C_VEL
LIN {X 0,Y 229.602,Z 615.371,A -85,B 0,C 180,E1 -20680.324,E2 -20680.324} C_VEL
LIN {X 0,Y 227.181,Z 616.292,A -85,B 0,C 180,E1 -20681.98,E2 -20681.98} C_VEL
LIN {X 0,Y 222.98,Z 616.909,A -85,B 0,C 180,E1 -20685.395,E2 -20685.395} C_VEL
LIN {X 0,Y 219.523,Z 615.927,A -85,B 0,C 180,E1 -20688.925,E2 -20688.925} C_VEL
LIN {X 0,Y 218.076,Z 614.849,A -85,B 0,C 180,E1 -20690.727,E2 -20690.727} C_VEL
LIN {X 0,Y 217.044,Z 613.314,A -85,B 0,C 180,E1 -20692.558,E2 -20692.558} C_VEL
LIN {X 0,Y 215.643,Z 610.269,A -85,B 0,C 180,E1 -20695.327,E2 -20695.327} C_VEL
LIN {X 0,Y 214.523,Z 606.244,A -85,B 0,C 180,E1 -20698.123,E2 -20698.123} C_VEL
LIN {X 0,Y 213.879,Z 601.149,A -85,B 0,C 180,E1 -20700.941,E2 -20700.941} C_VEL
LIN {X 0,Y 213.626,Z 593.61,A -85,B 0,C 180,E1 -20704.245,E2 -20704.245} C_VEL
LIN {X 0,Y 213.811,Z 585.633,A -85,B 0,C 180,E1 -20707.081,E2 -20707.081} C_VEL
LIN {X 0,Y 214.213,Z 577.654,A -85,B 0,C 180,E1 -20709.442,E2 -20709.442} C_VEL
LIN {X 0,Y 214.869,Z 567.132,A -85,B 0,C 180,E1 -20712.036,E2 -20712.036} C_VEL
LIN {X 0,Y 215.529,Z 556.644,A -85,B 0,C 180,E1 -20714.156,E2 -20714.156} C_VEL
LIN {X 0,Y 216.323,Z 543.695,A -85,B 0,C 180,E1 -20716.273,E2 -20716.273} C_VEL
LIN {X 0,Y 217.166,Z 530.109,A -85,B 0,C 180,E1 -20718.027,E2 -20718.027} C_VEL
LIN {X 0,Y 217.794,Z 517.249,A -85,B 0,C 180,E1 -20719.315,E2 -20719.315} C_VEL
LIN {X 0,Y 218.248,Z 502.698,A -85,B 0,C 180,E1 -20720.376,E2 -20720.376} C_VEL
LIN {X 0,Y 220.093,Z 446.048,A -85,B 0,C 180,E1 -20723.505,E2 -20723.505} C_VEL
LIN {X 0,Y 218.885,Z 440.949,A -85,B 0,C 180,E1 -20723.824,E2 -20723.824} C_VEL
LIN {X 0,Y 214.101,Z 422.993,A -85,B 0,C 180,E1 -20725.033,E2 -20725.033} C_VEL
LIN {X 0,Y 213.891,Z 421.975,A -85,B 0,C 180,E1 -20725.352,E2 -20725.352} C_VEL
LIN {X 0,Y 213.789,Z 421.843,A -85,B 0,C 180,E1 -20730.417,E2 -20730.417} C_VEL
LIN {X 0,Y 213.83,Z 422.257,A -85,B 0,C 180,E1 -20731.29,E2 -20731.29} C_VEL
LIN {X 0,Y 217.768,Z 430.91,A -85,B 0,C 180,E1 -20735.515,E2 -20735.515} C_VEL
LIN {X 0,Y 221.118,Z 438.724,A -85,B 0,C 180,E1 -20738.883,E2 -20738.883} C_VEL
LIN {X 0,Y 224.905,Z 449.141,A -85,B 0,C 180,E1 -20742.818,E2 -20742.818} C_VEL
LIN {X 0,Y 227.284,Z 456.42,A -85,B 0,C 180,E1 -20745.333,E2 -20745.333} C_VEL
LIN {X 0,Y 230.003,Z 466.46,A -85,B 0,C 180,E1 -20748.47,E2 -20748.47} C_VEL
LIN {X 0,Y 232.537,Z 478.158,A -85,B 0,C 180,E1 -20751.795,E2 -20751.795} C_VEL
LIN {X 0,Y 232.723,Z 481.087,A -85,B 0,C 180,E1 -20752.49,E2 -20752.49} C_VEL
LIN {X 0,Y 231.659,Z 488.41,A -85,B 0,C 180,E1 -20753.854,E2 -20753.854} C_VEL
LIN {X 0,Y 234.835,Z 512.537,A -85,B 0,C 180,E1 -20755.31,E2 -20755.31} C_VEL
LIN {X 0,Y 236.856,Z 530.624,A -85,B 0,C 180,E1 -20756.297,E2 -20756.297} C_VEL
LIN {X 0,Y 233.847,Z 601.164,A -85,B 0,C 180,E1 -20758.395,E2 -20758.395} C_VEL
LIN {X 0,Y 232.62,Z 613.767,A -85,B 0,C 180,E1 -20759.032,E2 -20759.032} C_VEL
LIN {X 0,Y 230.995,Z 625.972,A -85,B 0,C 180,E1 -20759.993,E2 -20759.993} C_VEL
LIN {X 0,Y 228.884,Z 638.313,A -85,B 0,C 180,E1 -20761.329,E2 -20761.329} C_VEL
LIN {X 0,Y 226.621,Z 648.664,A -85,B 0,C 180,E1 -20762.779,E2 -20762.779} C_VEL
LIN {X 0,Y 224.019,Z 659.272,A -85,B 0,C 180,E1 -20764.694,E2 -20764.694} C_VEL
LIN {X 0,Y 221.333,Z 669.476,A -85,B 0,C 180,E1 -20767.05,E2 -20767.05} C_VEL
LIN {X 0,Y 219.064,Z 677.373,A -85,B 0,C 180,E1 -20769.335,E2 -20769.335} C_VEL
LIN {X 0,Y 216.75,Z 684.859,A -85,B 0,C 180,E1 -20772.059,E2 -20772.059} C_VEL
LIN {X 0,Y 214.831,Z 690.866,A -85,B 0,C 180,E1 -20774.828,E2 -20774.828} C_VEL
LIN {X 0,Y 213.419,Z 695.616,A -85,B 0,C 180,E1 -20777.641,E2 -20777.641} C_VEL
LIN {X 0,Y 212.443,Z 699.249,A -85,B 0,C 180,E1 -20780.479,E2 -20780.479} C_VEL
LIN {X 0,Y 211.989,Z 701.119,A -85,B 0,C 180,E1 -20782.38,E2 -20782.38} C_VEL
LIN {X 0,Y 211.507,Z 703.222,A -85,B 0,C 180,E1 -20785.451,E2 -20785.451} C_VEL
LIN {X 0,Y 211.408,Z 704.159,A -85,B 0,C 180,E1 -20788.095,E2 -20788.095} C_VEL
LIN {X 0,Y 211.439,Z 704.391,A -85,B 0,C 180,E1 -20790,E2 -20790} C_VEL
LIN {X 0,Y 211.408,Z 704.193,A -85,B 0,C 180,E1 -20791.905,E2 -20791.905} C_VEL
LIN {X 0,Y 211.543,Z 703.23,A -85,B 0,C 180,E1 -20794.669,E2 -20794.669} C_VEL
LIN {X 0,Y 211.908,Z 701.242,A -85,B 0,C 180,E1 -20797.624,E2 -20797.624} C_VEL
LIN {X 0,Y 212.691,Z 698.343,A -85,B 0,C 180,E1 -20800.471,E2 -20800.471} C_VEL
LIN {X 0,Y 213.78,Z 694.405,A -85,B 0,C 180,E1 -20803.305,E2 -20803.305} C_VEL
LIN {X 0,Y 215.336,Z 689.301,A -85,B 0,C 180,E1 -20806.106,E2 -20806.106} C_VEL
LIN {X 0,Y 217.429,Z 682.868,A -85,B 0,C 180,E1 -20808.859,E2 -20808.859} C_VEL
LIN {X 0,Y 219.853,Z 674.875,A -85,B 0,C 180,E1 -20811.569,E2 -20811.569} C_VEL
LIN {X 0,Y 222.118,Z 666.703,A -85,B 0,C 180,E1 -20813.792,E2 -20813.792} C_VEL
LIN {X 0,Y 224.468,Z 657.766,A -85,B 0,C 180,E1 -20815.749,E2 -20815.749} C_VEL
LIN {X 0,Y 227.172,Z 646.682,A -85,B 0,C 180,E1 -20817.649,E2 -20817.649} C_VEL
LIN {X 0,Y 229.398,Z 635.868,A -85,B 0,C 180,E1 -20819.102,E2 -20819.102} C_VEL
LIN {X 0,Y 231.361,Z 623.912,A -85,B 0,C 180,E1 -20820.333,E2 -20820.333} C_VEL
LIN {X 0,Y 233.008,Z 611.471,A -85,B 0,C 180,E1 -20821.226,E2 -20821.226} C_VEL
LIN {X 0,Y 234.069,Z 598.835,A -85,B 0,C 180,E1 -20821.825,E2 -20821.825} C_VEL
LIN {X 0,Y 236.924,Z 530.476,A -85,B 0,C 180,E1 -20823.841,E2 -20823.841} C_VEL
LIN {X 0,Y 233.69,Z 502.458,A -85,B 0,C 180,E1 -20825.402,E2 -20825.402} C_VEL
LIN {X 0,Y 231.678,Z 487.949,A -85,B 0,C 180,E1 -20826.333,E2 -20826.333} C_VEL
LIN {X 0,Y 232.883,Z 479.592,A -85,B 0,C 180,E1 -20827.985,E2 -20827.985} C_VEL
LIN {X 0,Y 230.59,Z 468.648,A -85,B 0,C 180,E1 -20831.033,E2 -20831.033} C_VEL
LIN {X 0,Y 228.06,Z 458.956,A -85,B 0,C 180,E1 -20834.026,E2 -20834.026} C_VEL
LIN {X 0,Y 225.059,Z 449.549,A -85,B 0,C 180,E1 -20837.219,E2 -20837.219} C_VEL
LIN {X 0,Y 222.183,Z 441.497,A -85,B 0,C 180,E1 -20840.254,E2 -20840.254} C_VEL
LIN {X 0,Y 218.503,Z 432.572,A -85,B 0,C 180,E1 -20843.914,E2 -20843.914} C_VEL
LIN {X 0,Y 215.648,Z 426.052,A -85,B 0,C 180,E1 -20846.915,E2 -20846.915} C_VEL
LIN {X 0,Y 213.919,Z 422.729,A -85,B 0,C 180,E1 -20848.672,E2 -20848.672} C_VEL
LIN {X 0,Y 213.807,Z 421.87,A -85,B 0,C 180,E1 -20849.321,E2 -20849.321} C_VEL
LIN {X 0,Y 213.788,Z 421.843,A -85,B 0,C 180,E1 -20852.598,E2 -20852.598} C_VEL
LIN {X 0,Y 213.802,Z 421.83,A -85,B 0,C 180,E1 -20856.986,E2 -20856.986} C_VEL
LIN {X 0,Y 213.882,Z 421.816,A -85,B 0,C 180,E1 -20862.798,E2 -20862.798} C_VEL
LIN {X 0,Y 213.917,Z 421.82,A -85,B 0,C 180,E1 -20866.704,E2 -20866.704} C_VEL
LIN {X 0,Y 214.137,Z 421.793,A -85,B 0,C 180,E1 -20870.555,E2 -20870.555} C_VEL
LIN {X 0,Y 214.076,Z 421.788,A -85,B 0,C 180,E1 -20874.348,E2 -20874.348} C_VEL
LIN {X 0,Y 214.406,Z 421.771,A -85,B 0,C 180,E1 -20878.121,E2 -20878.121} C_VEL
LIN {X 0,Y 214.515,Z 421.753,A -85,B 0,C 180,E1 -20880,E2 -20880} C_VEL
LIN {X 0,Y 214.405,Z 421.742,A -85,B 0,C 180,E1 -20881.878,E2 -20881.878} C_VEL
LIN {X 0,Y 214.18,Z 421.789,A -85,B 0,C 180,E1 -20887.542,E2 -20887.542} C_VEL
LIN {X 0,Y 213.985,Z 421.806,A -85,B 0,C 180,E1 -20891.365,E2 -20891.365} C_VEL
LIN {X 0,Y 213.869,Z 421.818,A -85,B 0,C 180,E1 -20895.242,E2 -20895.242} C_VEL
LIN {X 0,Y 213.774,Z 421.847,A -85,B 0,C 180,E1 -20899.444,E2 -20899.444} C_VEL
LIN {X 0,Y 213.037,Z 421.936,A -85,B 0,C 180,E1 -20901.015,E2 -20901.015} C_VEL
